# B&R Automation Studio project 8238 (part 31)

### Program Logical/OPCuA_Client/Inwatec (IEC)

#### Variables.var
```iecst
VAR
	i : UINT;
	iw : REFERENCE TO Inwatec_typ;
	iw_d : REFERENCE TO Inwatec_data_typ;
	comm : REFERENCE TO Comm_typ;
	iw_r : REFERENCE TO Inwatec_data_typ;
END_VAR
```

#### Main.st
```iecst
PROGRAM _INIT
//Config and manage inwatec OPCuA communications
Inwatec[1].Config.ServerURL := 'opc.tcp://10.16.118.1:3001';
Inwatec[1].Config.Direction := INWATEC_RELEASE_TO;
Inwatec[1].Config.CommID 		:= 81;

Inwatec[2].Config.ServerURL := 'opc.tcp://10.16.118.1:3002';
Inwatec[2].Config.Direction := INWATEC_RELEASE_TO;
Inwatec[2].Config.CommID 		:= 82;

Inwatec[3].Config.ServerURL := 'opc.tcp://10.16.118.1:3003';
Inwatec[3].Config.Direction := INWATEC_RELEASE_TO;
Inwatec[3].Config.CommID 		:= 83;

Inwatec[4].Config.ServerURL := 'opc.tcp://10.16.118.1:3101';
Inwatec[4].Config.Direction := INWATEC_RECIEVE_FROM;
Inwatec[4].Config.CommID 		:= 84;

Inwatec[5].Config.ServerURL := 'opc.tcp://10.16.118.1:3102';
Inwatec[5].Config.Direction := INWATEC_RECIEVE_FROM;
Inwatec[5].Config.CommID 		:= 85;

Inwatec[6].Config.ServerURL := 'opc.tcp://10.16.118.1:3103';
Inwatec[6].Config.Direction := INWATEC_RECIEVE_FROM;
Inwatec[6].Config.CommID 		:= 86;

Inwatec[7].Config.ServerURL := 'opc.tcp://10.16.118.2:3001';
Inwatec[7].Config.Direction := INWATEC_RELEASE_TO;
Inwatec[7].Config.CommID 		:= 87;

Inwatec[8].Config.ServerURL := 'opc.tcp://10.16.118.2:3002';
Inwatec[8].Config.Direction := INWATEC_RELEASE_TO;
Inwatec[8].Config.CommID 		:= 88;

Inwatec[9].Config.ServerURL := 'opc.tcp://10.16.118.2:3003';
Inwatec[9].Config.Direction := INWATEC_RELEASE_TO;
Inwatec[9].Config.CommID 		:= 89;

Inwatec[10].Config.ServerURL := 'opc.tcp://10.16.118.2:3004';
Inwatec[10].Config.Direction := INWATEC_RELEASE_TO;
Inwatec[10].Config.CommID 		:= 90;

Inwatec[11].Config.ServerURL := 'opc.tcp://10.16.118.2:3101';
Inwatec[11].Config.Direction := INWATEC_RECIEVE_FROM;
Inwatec[11].Config.CommID 		:= 91;

END_PROGRAM

PROGRAM _CYCLIC

FOR i := 1 TO MAX_INWATEC_INTERFACES DO
	iw ACCESS ADR(Inwatec[i]);
	//Range check
	IF (iw.Config.CommID > 0) AND (iw.Config.CommID <= MAX_COMM) THEN
		comm ACCESS ADR(Comm[iw.Config.CommID]);

		CASE iw.Config.Direction OF
			INWATEC_RELEASE_TO:  // We need to set the batch information
				iw_d ACCESS ADR(iw.Outlet);		// Write Vars
				iw_r ACCESS ADR(iw.Inlet);		// Read Vars

				iw_d.batch_id 					:= comm.BatchID;
				iw_d.weight 						:= (UINT_TO_REAL(comm.Weight)/10);
				iw_d.customer_numeric 	:= comm.Customer;
				iw_d.category_numeric		:= comm.Category;
				iw_d.batch_count 				:= comm.Batch_QtyRemaining;

				iw_d.tx_handshake.0 		:= comm.BagReady;				// Bag in position

				// Read Variables
				comm.DropLoad 				:= iw_r.tx_handshake.0;
				comm.Unloading				:= iw_r.tx_handshake.1;
				comm.LoadDropped			:= iw_r.tx_handshake.2;

			INWATEC_RECIEVE_FROM:// We are reading the batch information.
				iw_d ACCESS ADR(iw.Inlet); 		// Write Vars
				iw_r ACCESS ADR(iw.Outlet);		// Read Vars

				iw_d.tx_handshake.0 		:= comm.ReadyToLoad; 	// Bag in position ready for load
				iw_d.tx_handshake.1 		:= comm.Loading;			// Recieving load
				iw_d.tx_handshake.2 		:= comm.LoadRecieved;	// Bag has recieved the load

				// Read Variables
				comm.BatchID 						:= iw_r.batch_id;
				comm.Weight							:= REAL_TO_UINT(iw_r.weight * 10);
				comm.Customer 					:= iw_r.customer_numeric;
				comm.Category						:= iw_r.category_numeric;
				comm.Batch_QtyRemaining	:= iw_r.batch_count;

				comm.ReadyToLoad				:= iw_r.tx_handshake.0;
				comm.Unloading					:= iw_r.tx_handshake.1;
				comm.UnloadFinished			:= iw_r.tx_handshake.2;

			ELSE
				iw_d ACCESS ADR(iw.Inlet);	// Code just ensure we don;t get a pointer error.
				iw_r ACCESS ADR(iw.Outlet);
		END_CASE;

		//Common controls.
		iw_d.system_status.0 := 0;// Is there any alarm on the device;
		iw_d.system_status.1 := 1; // PLC is alive;
		iw_d.system_status.2 := NOT comm.HaltSys; // System is in production (Maybe map Estop zone here)

		iw_d.i_am_alive 			:= Std.Clock1s;

		IF iw_r.i_am_alive THEN
			comm.LiveTime := 500; // 5s ish..
			iw_r.i_am_alive := 0;
		ELSIF (comm.LiveTime > 0) THEN
				comm.LiveTime := (comm.LiveTime - 1);
		END_IF;
		comm.Live := (comm.LiveTime > 0);

	END_IF;
END_FOR;

END_PROGRAM
```

### Program Logical/OPCuA_Client/OPCuAClient (IEC, version 1.00.1)

#### Main.st - Init, cyclic, exit code
```iecst
PROGRAM _INIT

	#if (MAX_OPCuA_CLIENTS < MAX_INWATEC_INTERFACES)
		#error 'Not enough opcua clients for Inwatec'
	#endif

	_inwatec_config;

	////Test connection.
	//OPCuA_Client[3].Config.ServerURL :=	'opc.tcp://10.8.4.20:4840';  // IP Address of interface.
	//
	//OPCuA_Client[3].Config.SessionUser.UserIdentityTokenType := UAUITT_Username;
	//OPCuA_Client[3].Config.SessionUser.TokenParam1 := 'test';  //UserName
	//OPCuA_Client[3].Config.SessionUser.TokenParam2 := 'test';  //Password
	//
	//
	////Set the Vars.
	//OPCuA_Client[3].Config.Data.Read[0].NodeID.Identifier := '::AsGlobalPV:OpcUa.VC[231].Write.Heartbeat';
	//OPCuA_Client[3].Config.Data.Read[0].Variable := 'TestRead[0]';
	//OPCuA_Client[3].Config.Data.Read[1].NodeID.Identifier := '::AsGlobalPV:OpcUa.VC[231].Write.PermissionToMove';
	//OPCuA_Client[3].Config.Data.Read[1].Variable := 'TestRead[1]';
	//OPCuA_Client[3].Config.Data.Read[2].NodeID.Identifier := '::AsGlobalPV:OpcUa.VC[231].Write.ReleaseBag';
	//OPCuA_Client[3].Config.Data.Read[2].Variable := 'TestRead[2]';
	//OPCuA_Client[3].Config.Data.Read[3].NodeID.Identifier := '::AsGlobalPV:OpcUa.VC[231].Write.ReceiveBag';
	//OPCuA_Client[3].Config.Data.Read[3].Variable := 'TestRead[3]';
	//
	//OPCuA_Client[3].Config.Data.Write[0].NodeID.Identifier := '::AsGlobalPV:OpcUa.VC[231].Read.Heartbeat';
	//OPCuA_Client[3].Config.Data.Write[0].Variable := 'TestWrite[0]';
	//OPCuA_Client[3].Config.Data.Write[1].NodeID.Identifier := '::AsGlobalPV:OpcUa.VC[231].Read.Auto';
	//OPCuA_Client[3].Config.Data.Write[1].Variable := 'TestWrite[1]';
	//OPCuA_Client[3].Config.Data.Write[2].NodeID.Identifier := '::AsGlobalPV:OpcUa.VC[231].Read.Manual';
	//OPCuA_Client[3].Config.Data.Write[2].Variable := 'TestWrite[2]';
	//OPCuA_Client[3].Config.Data.Write[3].NodeID.Identifier := '::AsGlobalPV:OpcUa.VC[231].Read.ChuteBlocked';
	//OPCuA_Client[3].Config.Data.Write[3].Variable := 'TestWrite[3]';

	FOR x := 1 TO MAX_OPCuA_CLIENTS DO
		client ACCESS ADR (OPCuA_Client[x]);
		client.Config.SessionInfo.SessionName := 'supertrack';
		client.Config.SessionInfo.ApplicationName := '';
		client.Config.SessionInfo.SecurityMsgMode := UASecurityMsgMode_Sign;//UASecurityMsgMode_BestAvailab;
		client.Config.SessionInfo.SecurityPolicy := UASecurityPolicy_Basic256Sha256;//UASecurityPolicy_BestAvailable;
		client.Config.SessionInfo.CertificateStore := '';
		client.Config.SessionInfo.ClientCertificateName := '';
		client.Config.SessionInfo.ServerUri := '';
		client.Config.SessionInfo.CheckServerCertificate := 0;
		client.Config.SessionInfo.TransportProfile := UATP_UATcp;
		client.Config.SessionInfo.UserIdentityToken := client.Config.SessionUser;
		client.Config.SessionInfo.VendorSpecificParameter := '';
		client.Config.SessionInfo.SessionTimeout := T#5s;
		client.Config.SessionInfo.MonitorConnection := T#500ms;
		//client.Config.SessionInfo.LocaleIDs

		client.Config.Data.ReadCount := MAX_READ_NODES;
		FOR i := 0 TO MAX_READ_NODES DO
			client.Config.Data.Read[i].NodeID.IdentifierType := UAIdentifierType_String;
			client.Config.Data.Read[i].NodeInfo.AttributeId := UAAI_Value;
			IF (client.Config.Data.Read[i].NodeID.Identifier = '') THEN
				client.Config.Data.ReadCount := i;
				EXIT;
			END_IF;
		END_FOR;

		client.Config.Data.WriteCount := MAX_WRITE_NODES;
		FOR i := 0 TO MAX_WRITE_NODES DO
			client.Config.Data.Write[i].NodeID.IdentifierType := UAIdentifierType_String;
			client.Config.Data.Write[i].NodeInfo.AttributeId := UAAI_Value;
			IF (client.Config.Data.Write[i].NodeID.Identifier = '') THEN
				client.Config.Data.WriteCount := i;
				EXIT;
			END_IF;
		END_FOR;

		client.Functions.RetryTimer.PT := T#5s; // Time to try to reconnect if the server isn;t available.
	END_FOR;

END_PROGRAM

PROGRAM _CYCLIC
//MAX of 40 Connections.

	FOR x := 1 TO MAX_OPCuA_CLIENTS DO
		client ACCESS ADR (OPCuA_Client[x]);
		f ACCESS ADR(client.Functions);
		IF client.Config.ServerURL <> '' THEN

			f.Connect.Execute 			:= (client.State = OPCuA_CLIENT_STATE_CONNECT);
			f.GetNameSpace.Execute	:= (client.State = OPCuA_CLIENT_STATE_GET_NAMESPACE);
			f.ReadBulk.Execute := f.WriteBulk.Execute	:= (client.State = OPCuA_CLIENT_STATE_READ_WRITE);
			f.Disconnect.Execute 		:= (client.State = OPCuA_CLIENT_STATE_DISCONNECT);

			CASE client.State OF

				OPCuA_CLIENT_STATE_CONNECT:
					f.Connect.ServerEndpointUrl := client.Config.ServerURL;
					f.Connect.SessionConnectInfo := client.Config.SessionInfo;
					f.Connect.Timeout := T#1s;
					IF f.Connect.Done THEN
						client.State := OPCuA_CLIENT_STATE_GET_NAMESPACE;
					ELSIF f.Connect.Error THEN
						client.Error.ErrorState := client.State;
						client.State := OPCuA_CLIENT_STATE_ERROR;
						client.Error.ErrorID :=  f.Connect.ErrorID;
					END_IF;

				OPCuA_CLIENT_STATE_GET_NAMESPACE:
					f.GetNameSpace.ConnectionHdl  := f.Connect.ConnectionHdl;
					f.GetNameSpace.NamespaceUri		:= 'urn:B&R/pv/';
					f.GetNameSpace.Timeout 				:= T#1s;

					IF f.GetNameSpace.Done THEN
						client.State := OPCuA_CLIENT_STATE_BUILD_DATA;
					ELSIF f.GetNameSpace.Error THEN
						client.Error.ErrorState := client.State;
						client.State := OPCuA_CLIENT_STATE_ERROR;
						client.Error.ErrorID :=  f.GetNameSpace.ErrorID;
					END_IF;

				OPCuA_CLIENT_STATE_BUILD_DATA:

					FOR i := 0 TO client.Config.Data.ReadCount DO
						client.ReadData.NodeID[i].NamespaceIndex 	:= f.GetNameSpace.NamespaceIndex;
						client.ReadData.NodeID[i].IdentifierType 	:= client.Config.Data.Read[i].NodeID.IdentifierType;
						client.ReadData.NodeID[i].Identifier 			:= client.Config.Data.Read[i].NodeID.Identifier;
						client.ReadData.NodeInfo[i].AttributeId 	:= client.Config.Data.Read[i].NodeInfo.AttributeId;
						client.ReadData.Variable[i]								:= client.Config.Data.Read[i].Variable;
					END_FOR;

					FOR i := 0 TO client.Config.Data.WriteCount DO
						client.WriteData.NodeID[i].NamespaceIndex 	:= f.GetNameSpace.NamespaceIndex;
						client.WriteData.NodeID[i].IdentifierType 	:= client.Config.Data.Write[i].NodeID.IdentifierType;
						client.WriteData.NodeID[i].Identifier 			:= client.Config.Data.Write[i].NodeID.Identifier;
						client.WriteData.NodeInfo[i].AttributeId 		:= client.Config.Data.Write[i].NodeInfo.AttributeId;
						client.WriteData.Variable[i]								:= client.Config.Data.Write[i].Variable;

					END_FOR;

					client.State := OPCuA_CLIENT_STATE_READ_WRITE;

				OPCuA_CLIENT_STATE_READ_WRITE:
					f.ReadBulk.ConnectionHdl 	:= f.Connect.ConnectionHdl;
					f.ReadBulk.NodeIDCount 		:= client.Config.Data.ReadCount;
					f.ReadBulk.NodeAddInfo 		:= ADR(client.ReadData.NodeInfo);
					f.ReadBulk.NodeErrorIDs 	:= ADR(client.ReadData.ErrorID);
					f.ReadBulk.NodeIDs 				:= ADR(client.ReadData.NodeID);
					f.ReadBulk.TimeStamps 		:= ADR(client.ReadData.TimeStamps);
					f.ReadBulk.Variables 			:= ADR(client.ReadData.Variable);
					f.ReadBulk.Timeout 				:= T#1500ms;
					IF f.ReadBulk.Done THEN
						f.ReadBulk.Execute := 0; // Read Cyclica
						f.ReadBulk;
					ELSIF f.ReadBulk.Error THEN
						IF 	f.ReadBulk.ErrorID = OPCuA_ERR_OUT_OF_SERVICE THEN
							client.State := OPCuA_CLIENT_STATE_DISCONNECT;
						ELSE
							client.Error.ErrorState := client.State;
							client.State := OPCuA_CLIENT_STATE_ERROR;
							IF (f.ReadBulk.ErrorID > 0) THEN
								client.Error.ErrorID := f.ReadBulk.ErrorID;
							ELSE
								//Look for the bad node..
								FOR i := 0 TO client.Config.Data.ReadCount DO
									IF (client.ReadData.ErrorID[i] > 0) THEN
										client.Error.ErrorID := client.ReadData.ErrorID[i];
										client.Error.ErrorNode := i;
										EXIT;
									END_IF;
								END_FOR;
							END_IF;
						END_IF;

					END_IF

					//Disadvantage of writing like this, is we are always pushing just like tradional TCP.
					f.WriteBulk.ConnectionHdl := f.Connect.ConnectionHdl;
					f.WriteBulk.NodeIDCount		:= client.Config.Data.WriteCount;
					f.WriteBulk.NodeAddInfo		:= ADR(client.WriteData.NodeInfo);
					f.WriteBulk.NodeErrorIDs	:= ADR(client.WriteData.ErrorID);
					f.WriteBulk.NodeIDs				:= ADR(client.WriteData.NodeID);
					f.WriteBulk.Variables			:= ADR(client.WriteData.Variable);
					f.WriteBulk.Timeout				:= T#1500ms;

					IF f.WriteBulk.Done THEN
						f.WriteBulk.Execute := 0; // Read Cyclica
						f.WriteBulk();
					ELSIF f.WriteBulk.Error THEN
						IF 	f.WriteBulk.ErrorID = OPCuA_ERR_OUT_OF_SERVICE THEN
							client.State := OPCuA_CLIENT_STATE_DISCONNECT;
						ELSE
							client.Error.ErrorState := OPCuA_CLIENT_STATE_READ_WRITE + 1000;// Add 1000 to show its a write failure.
							client.State := OPCuA_CLIENT_STATE_ERROR;
							IF (f.WriteBulk.ErrorID > 0) THEN
								client.Error.ErrorID := f.WriteBulk.ErrorID;
							ELSE
								//Look for the bad node..
								FOR i := 0 TO client.Config.Data.WriteCount DO
									IF (client.WriteData.ErrorID[i] > 0) THEN
										client.Error.ErrorID := client.WriteData.ErrorID[i];
										client.Error.ErrorNode := i;
										EXIT;
									END_IF;
								END_FOR;
							END_IF;
						END_IF;

					END_IF;

				OPCuA_CLIENT_STATE_DISCONNECT:
					f.Disconnect.ConnectionHdl := f.Connect.ConnectionHdl;
					f.Disconnect.Timeout := T#2s;
					IF f.Disconnect.Done THEN
						client.State := OPCuA_CLIENT_STATE_CONNECT;
					ELSIF f.Disconnect.Error THEN
						IF (f.Connect.ConnectionHdl = 0) OR (f.Disconnect.ErrorID = 16#A0080000) OR (f.Disconnect.ErrorID = 16#80AD0000)  THEN
							client.State := OPCuA_CLIENT_STATE_CONNECT;
						ELSE
							//client.State := OPCuA_CLIENT_STATE_ERROR;
							//client.Error.ErrorID := f.Disconnect.ErrorID;
						END_IF;
					END_IF;

				OPCuA_CLIENT_STATE_ERROR:
					//Maybe should just write to a logger then restart!
					IF client.Functions.RetryTimer.Q THEN
						IF (f.Connect.ConnectionHdl > 0) THEN
							client.State := OPCuA_CLIENT_STATE_DISCONNECT; // Always try to disconnect any open connections before reconnecting.
						ELSE
							client.State := OPCuA_CLIENT_STATE_CONNECT;
						END_IF;
					ELSIF (client.Error.ErrorID = OPCuA_ERR_TIMEOUT) THEN
						//				client.Functions.RetryTimer.IN := 1;
						//			ELSE
						//				client.State := OPCuA_CLIENT_STATE_DISCONNECT;
					END_IF;

			END_CASE;
			client.Functions.ErrorStatePLS.CLK := (client.State = OPCuA_CLIENT_STATE_ERROR);
			client.Functions.ErrorStatePLS();

			IF client.Functions.ErrorStatePLS.Q THEN
				brsmemcpy(ADR(client.Error.ErrorCode),ADR(client.Error.ErrorID) + 2,2);
				getErrorText.ErrorID := client.Error.ErrorCode;
				getErrorText();
				client.Error.Message := 	getErrorText.ErrorMessage;
			END_IF;

			f.Connect();
			f.GetNameSpace();
			f.ReadBulk();
			f.WriteBulk();
			f.Disconnect();
			client.Functions.RetryTimer.IN := (client.State = OPCuA_CLIENT_STATE_ERROR);
			client.Functions.RetryTimer();
		//client.Functions.RetryTimer.IN := 0;
		END_IF;
	END_FOR;
	//TestRead;//
	//TestWrite;
	//	TestReadx;//
	//	TestWritex;

END_PROGRAM

PROGRAM _EXIT
(* Insert code here *)

END_PROGRAM
```

#### inwatec.st - *Special config for building inwatec interfaces
```iecst
ACTION _inwatec_config:

FOR i := 1 TO MAX_INWATEC_INTERFACES DO
	//Always match the inwatec array to the opcua array
	iw ACCESS ADR(Inwatec[i]);
	client ACCESS ADR(OPCuA_Client[i]);

	client.Config.ServerURL :=	iw.Config.ServerURL;
	client.Config.SessionUser := iw.Config.Authenication;

	CASE iw.Config.Direction OF
		0: //Dropping onto Inwatec
			//Write to Outlet, Read from Inlet

			client.Config.Data.Read[0].NodeID.Identifier := '::BatchIn:batch_to_inwatec[0].inlet.batch_count';
			client.Config.Data.Read[1].NodeID.Identifier := '::BatchIn:batch_to_inwatec[0].inlet.batch_id';
			client.Config.Data.Read[2].NodeID.Identifier := '::BatchIn:batch_to_inwatec[0].inlet.category';
			client.Config.Data.Read[3].NodeID.Identifier := '::BatchIn:batch_to_inwatec[0].inlet.category_name';
			client.Config.Data.Read[4].NodeID.Identifier := '::BatchIn:batch_to_inwatec[0].inlet.category_numeric';
			client.Config.Data.Read[5].NodeID.Identifier := '::BatchIn:batch_to_inwatec[0].inlet.customer';
			client.Config.Data.Read[6].NodeID.Identifier := '::BatchIn:batch_to_inwatec[0].inlet.customer_name';
			client.Config.Data.Read[7].NodeID.Identifier := '::BatchIn:batch_to_inwatec[0].inlet.customer_numeric';
			client.Config.Data.Read[8].NodeID.Identifier := '::BatchIn:batch_to_inwatec[0].inlet.i_am_alive';
			client.Config.Data.Read[9].NodeID.Identifier := '::BatchIn:batch_to_inwatec[0].inlet.lot';
			client.Config.Data.Read[10].NodeID.Identifier := '::BatchIn:batch_to_inwatec[0].inlet.lot_numeric';
			client.Config.Data.Read[11].NodeID.Identifier := '::BatchIn:batch_to_inwatec[0].inlet.option_1';
			client.Config.Data.Read[12].NodeID.Identifier := '::BatchIn:batch_to_inwatec[0].inlet.option_2';
			client.Config.Data.Read[13].NodeID.Identifier := '::BatchIn:batch_to_inwatec[0].inlet.source_id';
			client.Config.Data.Read[14].NodeID.Identifier := '::BatchIn:batch_to_inwatec[0].inlet.sublot';
			client.Config.Data.Read[15].NodeID.Identifier := '::BatchIn:batch_to_inwatec[0].inlet.sublot_numeric';
			client.Config.Data.Read[16].NodeID.Identifier := '::BatchIn:batch_to_inwatec[0].inlet.system_status';
			client.Config.Data.Read[17].NodeID.Identifier := '::BatchIn:batch_to_inwatec[0].inlet.tx_handshake';
			client.Config.Data.Read[18].NodeID.Identifier := '::BatchIn:batch_to_inwatec[0].inlet.weight';
			client.Config.Data.Read[19].NodeID.Identifier := '::BatchIn:batch_to_inwatec[0].inlet.option_flag_1';
			client.Config.Data.Read[20].NodeID.Identifier := '::BatchIn:batch_to_inwatec[0].inlet.option_flag_2';

			client.Config.Data.Write[0].NodeID.Identifier := '::BatchIn:batch_to_inwatec[0].outlet.batch_count';
			client.Config.Data.Write[1].NodeID.Identifier := '::BatchIn:batch_to_inwatec[0].outlet.batch_id';
			client.Config.Data.Write[2].NodeID.Identifier := '::BatchIn:batch_to_inwatec[0].outlet.category';
			client.Config.Data.Write[3].NodeID.Identifier := '::BatchIn:batch_to_inwatec[0].outlet.category_name';
			client.Config.Data.Write[4].NodeID.Identifier := '::BatchIn:batch_to_inwatec[0].outlet.category_numeric';
			client.Config.Data.Write[5].NodeID.Identifier := '::BatchIn:batch_to_inwatec[0].outlet.customer';
			client.Config.Data.Write[6].NodeID.Identifier := '::BatchIn:batch_to_inwatec[0].outlet.customer_name';
			client.Config.Data.Write[7].NodeID.Identifier := '::BatchIn:batch_to_inwatec[0].outlet.customer_numeric';
			client.Config.Data.Write[8].NodeID.Identifier := '::BatchIn:batch_to_inwatec[0].outlet.i_am_alive';
			client.Config.Data.Write[9].NodeID.Identifier := '::BatchIn:batch_to_inwatec[0].outlet.lot';
			client.Config.Data.Write[10].NodeID.Identifier := '::BatchIn:batch_to_inwatec[0].outlet.lot_numeric';
			client.Config.Data.Write[11].NodeID.Identifier := '::BatchIn:batch_to_inwatec[0].outlet.option_1';
			client.Config.Data.Write[12].NodeID.Identifier := '::BatchIn:batch_to_inwatec[0].outlet.option_2';
			client.Config.Data.Write[13].NodeID.Identifier := '::BatchIn:batch_to_inwatec[0].outlet.source_id';
			client.Config.Data.Write[14].NodeID.Identifier := '::BatchIn:batch_to_inwatec[0].outlet.sublot';
			client.Config.Data.Write[15].NodeID.Identifier := '::BatchIn:batch_to_inwatec[0].outlet.sublot_numeric';
			client.Config.Data.Write[16].NodeID.Identifier := '::BatchIn:batch_to_inwatec[0].outlet.system_status';
			client.Config.Data.Write[17].NodeID.Identifier := '::BatchIn:batch_to_inwatec[0].outlet.tx_handshake';
			client.Config.Data.Write[18].NodeID.Identifier := '::BatchIn:batch_to_inwatec[0].outlet.weight';
			client.Config.Data.Write[19].NodeID.Identifier := '::BatchIn:batch_to_inwatec[0].outlet.option_flag_1';
			client.Config.Data.Write[20].NodeID.Identifier := '::BatchIn:batch_to_inwatec[0].outlet.option_flag_2';

			brsitoa(i,ADR(str_index));
			FOR x := 0 TO MAX_READ_NODES DO
				client.Config.Data.Read[x].Variable := 'Inwatec[';
				brsstrcat(ADR(client.Config.Data.Read[x].Variable),ADR(str_index));
			END_FOR;
			brsstrcat(ADR(client.Config.Data.Read[0].Variable),ADR('].Inlet.batch_count'));
			brsstrcat(ADR(client.Config.Data.Read[1].Variable),ADR('].Inlet.batch_id'));
			brsstrcat(ADR(client.Config.Data.Read[2].Variable),ADR('].Inlet.category'));
			brsstrcat(ADR(client.Config.Data.Read[3].Variable),ADR('].Inlet.category_name'));
			brsstrcat(ADR(client.Config.Data.Read[4].Variable),ADR('].Inlet.category_numeric'));
			brsstrcat(ADR(client.Config.Data.Read[5].Variable),ADR('].Inlet.customer'));
			brsstrcat(ADR(client.Config.Data.Read[6].Variable),ADR('].Inlet.customer_name'));
			brsstrcat(ADR(client.Config.Data.Read[7].Variable),ADR('].Inlet.customer_numeric'));
			brsstrcat(ADR(client.Config.Data.Read[8].Variable),ADR('].Inlet.i_am_alive'));
			brsstrcat(ADR(client.Config.Data.Read[9].Variable),ADR('].Inlet.lot'));
			brsstrcat(ADR(client.Config.Data.Read[10].Variable),ADR('].Inlet.lot_numeric'));
			brsstrcat(ADR(client.Config.Data.Read[11].Variable),ADR('].Inlet.option_1'));
			brsstrcat(ADR(client.Config.Data.Read[12].Variable),ADR('].Inlet.option_2'));
			brsstrcat(ADR(client.Config.Data.Read[13].Variable),ADR('].Inlet.source_id'));
			brsstrcat(ADR(client.Config.Data.Read[14].Variable),ADR('].Inlet.sublot'));
			brsstrcat(ADR(client.Config.Data.Read[15].Variable),ADR('].Inlet.sublot_numeric'));
			brsstrcat(ADR(client.Config.Data.Read[16].Variable),ADR('].Inlet.system_status'));
			brsstrcat(ADR(client.Config.Data.Read[17].Variable),ADR('].Inlet.tx_handshake'));
			brsstrcat(ADR(client.Config.Data.Read[18].Variable),ADR('].Inlet.weight'));
			brsstrcat(ADR(client.Config.Data.Read[19].Variable),ADR('].Inlet.option_flag_1'));
			brsstrcat(ADR(client.Config.Data.Read[20].Variable),ADR('].Inlet.option_flag_2'));

			brsitoa(i,ADR(str_index));
			FOR x := 0 TO MAX_WRITE_NODES DO
				client.Config.Data.Read[x].Variable := 'Inwatec[';
				brsstrcat(ADR(client.Config.Data.Read[x].Variable),ADR(str_index));
			END_FOR;
			brsstrcat(ADR(client.Config.Data.Write[0].Variable),ADR('].Outlet.batch_count'));
			brsstrcat(ADR(client.Config.Data.Write[1].Variable),ADR('].Outlet.batch_id'));
			brsstrcat(ADR(client.Config.Data.Write[2].Variable),ADR('].Outlet.category'));
			brsstrcat(ADR(client.Config.Data.Write[3].Variable),ADR('].Outlet.category_name'));
			brsstrcat(ADR(client.Config.Data.Write[4].Variable),ADR('].Outlet.category_numeric'));
			brsstrcat(ADR(client.Config.Data.Write[5].Variable),ADR('].Outlet.customer'));
			brsstrcat(ADR(client.Config.Data.Write[6].Variable),ADR('].Outlet.customer_name'));
			brsstrcat(ADR(client.Config.Data.Write[7].Variable),ADR('].Outlet.customer_numeric'));
			brsstrcat(ADR(client.Config.Data.Write[8].Variable),ADR('].Outlet.i_am_alive'));
			brsstrcat(ADR(client.Config.Data.Write[9].Variable),ADR('].Outlet.lot'));
			brsstrcat(ADR(client.Config.Data.Write[10].Variable),ADR('].Outlet.lot_numeric'));
			brsstrcat(ADR(client.Config.Data.Write[11].Variable),ADR('].Outlet.option_1'));
			brsstrcat(ADR(client.Config.Data.Write[12].Variable),ADR('].Outlet.option_2'));
			brsstrcat(ADR(client.Config.Data.Write[13].Variable),ADR('].Outlet.source_id'));
			brsstrcat(ADR(client.Config.Data.Write[14].Variable),ADR('].Outlet.sublot'));
			brsstrcat(ADR(client.Config.Data.Write[15].Variable),ADR('].Outlet.sublot_numeric'));
			brsstrcat(ADR(client.Config.Data.Write[16].Variable),ADR('].Outlet.system_status'));
			brsstrcat(ADR(client.Config.Data.Write[17].Variable),ADR('].Outlet.tx_handshake'));
			brsstrcat(ADR(client.Config.Data.Write[18].Variable),ADR('].Outlet.weight'));
			brsstrcat(ADR(client.Config.Data.Write[19].Variable),ADR('].Outlet.option_flag_1'));
			brsstrcat(ADR(client.Config.Data.Write[20].Variable),ADR('].Outlet.option_flag_2'));

		1: //Recieving from Inwatec
				//Write to Inlet, Read from Outlet
				client.Config.Data.Read[0].NodeID.Identifier := '::BatchOut:batch_from_inwatec[0].outlet.batch_count';
				client.Config.Data.Read[1].NodeID.Identifier := '::BatchOut:batch_from_inwatec[0].outlet.batch_id';
				client.Config.Data.Read[2].NodeID.Identifier := '::BatchOut:batch_from_inwatec[0].outlet.category';
				client.Config.Data.Read[3].NodeID.Identifier := '::BatchOut:batch_from_inwatec[0].outlet.category_name';
				client.Config.Data.Read[4].NodeID.Identifier := '::BatchOut:batch_from_inwatec[0].outlet.category_numeric';
				client.Config.Data.Read[5].NodeID.Identifier := '::BatchOut:batch_from_inwatec[0].outlet.customer';
				client.Config.Data.Read[6].NodeID.Identifier := '::BatchOut:batch_from_inwatec[0].outlet.customer_name';
				client.Config.Data.Read[7].NodeID.Identifier := '::BatchOut:batch_from_inwatec[0].outlet.customer_numeric';
				client.Config.Data.Read[8].NodeID.Identifier := '::BatchOut:batch_from_inwatec[0].outlet.i_am_alive';
				client.Config.Data.Read[9].NodeID.Identifier := '::BatchOut:batch_from_inwatec[0].outlet.lot';
				client.Config.Data.Read[10].NodeID.Identifier := '::BatchOut:batch_from_inwatec[0].outlet.lot_numeric';
				client.Config.Data.Read[11].NodeID.Identifier := '::BatchOut:batch_from_inwatec[0].outlet.option_1';
				client.Config.Data.Read[12].NodeID.Identifier := '::BatchOut:batch_from_inwatec[0].outlet.option_2';
				client.Config.Data.Read[13].NodeID.Identifier := '::BatchOut:batch_from_inwatec[0].outlet.source_id';
				client.Config.Data.Read[14].NodeID.Identifier := '::BatchOut:batch_from_inwatec[0].outlet.sublot';
				client.Config.Data.Read[15].NodeID.Identifier := '::BatchOut:batch_from_inwatec[0].outlet.sublot_numeric';
				client.Config.Data.Read[16].NodeID.Identifier := '::BatchOut:batch_from_inwatec[0].outlet.system_status';
				client.Config.Data.Read[17].NodeID.Identifier := '::BatchOut:batch_from_inwatec[0].outlet.tx_handshake';
				client.Config.Data.Read[18].NodeID.Identifier := '::BatchOut:batch_from_inwatec[0].outlet.weight';
				client.Config.Data.Read[19].NodeID.Identifier := '::BatchOut:batch_from_inwatec[0].outlet.option_flag_1';
				client.Config.Data.Read[20].NodeID.Identifier := '::BatchOut:batch_from_inwatec[0].outlet.option_flag_2';

				client.Config.Data.Write[0].NodeID.Identifier := '::BatchOut:batch_from_inwatec[0].inlet.batch_count';
				client.Config.Data.Write[1].NodeID.Identifier := '::BatchOut:batch_from_inwatec[0].inlet.batch_id';
				client.Config.Data.Write[2].NodeID.Identifier := '::BatchOut:batch_from_inwatec[0].inlet.category';
				client.Config.Data.Write[3].NodeID.Identifier := '::BatchOut:batch_from_inwatec[0].inlet.category_name';
				client.Config.Data.Write[4].NodeID.Identifier := '::BatchOut:batch_from_inwatec[0].inlet.category_numeric';
				client.Config.Data.Write[5].NodeID.Identifier := '::BatchOut:batch_from_inwatec[0].inlet.customer';
				client.Config.Data.Write[6].NodeID.Identifier := '::BatchOut:batch_from_inwatec[0].inlet.customer_name';
				client.Config.Data.Write[7].NodeID.Identifier := '::BatchOut:batch_from_inwatec[0].inlet.customer_numeric';
				client.Config.Data.Write[8].NodeID.Identifier := '::BatchOut:batch_from_inwatec[0].inlet.i_am_alive';
				client.Config.Data.Write[9].NodeID.Identifier := '::BatchOut:batch_from_inwatec[0].inlet.lot';
				client.Config.Data.Write[10].NodeID.Identifier := '::BatchOut:batch_from_inwatec[0].inlet.lot_numeric';
				client.Config.Data.Write[11].NodeID.Identifier := '::BatchOut:batch_from_inwatec[0].inlet.option_1';
				client.Config.Data.Write[12].NodeID.Identifier := '::BatchOut:batch_from_inwatec[0].inlet.option_2';
				client.Config.Data.Write[13].NodeID.Identifier := '::BatchOut:batch_from_inwatec[0].inlet.source_id';
				client.Config.Data.Write[14].NodeID.Identifier := '::BatchOut:batch_from_inwatec[0].inlet.sublot';
				client.Config.Data.Write[15].NodeID.Identifier := '::BatchOut:batch_from_inwatec[0].inlet.sublot_numeric';
				client.Config.Data.Write[16].NodeID.Identifier := '::BatchOut:batch_from_inwatec[0].inlet.system_status';
				client.Config.Data.Write[17].NodeID.Identifier := '::BatchOut:batch_from_inwatec[0].inlet.tx_handshake';
				client.Config.Data.Write[18].NodeID.Identifier := '::BatchOut:batch_from_inwatec[0].inlet.weight';
				client.Config.Data.Write[19].NodeID.Identifier := '::BatchOut:batch_from_inwatec[0].inlet.option_flag_1';
				client.Config.Data.Write[20].NodeID.Identifier := '::BatchOut:batch_from_inwatec[0].inlet.option_flag_2';

				brsitoa(i,ADR(str_index));
				FOR x := 0 TO MAX_READ_NODES DO
					client.Config.Data.Read[x].Variable := 'Inwatec[';
					brsstrcat(ADR(client.Config.Data.Read[x].Variable),ADR(str_index));
				END_FOR;
				brsstrcat(ADR(client.Config.Data.Read[0].Variable),ADR('].Outlet.batch_count'));
				brsstrcat(ADR(client.Config.Data.Read[1].Variable),ADR('].Outlet.batch_id'));
				brsstrcat(ADR(client.Config.Data.Read[2].Variable),ADR('].Outlet.category'));
				brsstrcat(ADR(client.Config.Data.Read[3].Variable),ADR('].Outlet.category_name'));
				brsstrcat(ADR(client.Config.Data.Read[4].Variable),ADR('].Outlet.category_numeric'));
				brsstrcat(ADR(client.Config.Data.Read[5].Variable),ADR('].Outlet.customer'));
				brsstrcat(ADR(client.Config.Data.Read[6].Variable),ADR('].Outlet.customer_name'));
				brsstrcat(ADR(client.Config.Data.Read[7].Variable),ADR('].Outlet.customer_numeric'));
				brsstrcat(ADR(client.Config.Data.Read[8].Variable),ADR('].Outlet.i_am_alive'));
				brsstrcat(ADR(client.Config.Data.Read[9].Variable),ADR('].Outlet.lot'));
				brsstrcat(ADR(client.Config.Data.Read[10].Variable),ADR('].Outlet.lot_numeric'));
				brsstrcat(ADR(client.Config.Data.Read[11].Variable),ADR('].Outlet.option_1'));
				brsstrcat(ADR(client.Config.Data.Read[12].Variable),ADR('].Outlet.option_2'));
				brsstrcat(ADR(client.Config.Data.Read[13].Variable),ADR('].Outlet.source_id'));
				brsstrcat(ADR(client.Config.Data.Read[14].Variable),ADR('].Outlet.sublot'));
				brsstrcat(ADR(client.Config.Data.Read[15].Variable),ADR('].Outlet.sublot_numeric'));
				brsstrcat(ADR(client.Config.Data.Read[16].Variable),ADR('].Outlet.system_status'));
				brsstrcat(ADR(client.Config.Data.Read[17].Variable),ADR('].Outlet.tx_handshake'));
				brsstrcat(ADR(client.Config.Data.Read[18].Variable),ADR('].Outlet.weight'));
				brsstrcat(ADR(client.Config.Data.Read[19].Variable),ADR('].Outlet.option_flag_1'));
				brsstrcat(ADR(client.Config.Data.Read[20].Variable),ADR('].Outlet.option_flag_2'));

				brsitoa(i,ADR(str_index));
				FOR x := 0 TO MAX_WRITE_NODES DO
					client.Config.Data.Read[x].Variable := 'Inwatec[';
					brsstrcat(ADR(client.Config.Data.Read[x].Variable),ADR(str_index));
				END_FOR;
				brsstrcat(ADR(client.Config.Data.Write[0].Variable),ADR('].Inlet.batch_count'));
				brsstrcat(ADR(client.Config.Data.Write[1].Variable),ADR('].Inlet.batch_id'));
				brsstrcat(ADR(client.Config.Data.Write[2].Variable),ADR('].Inlet.category'));
				brsstrcat(ADR(client.Config.Data.Write[3].Variable),ADR('].Inlet.category_name'));
				brsstrcat(ADR(client.Config.Data.Write[4].Variable),ADR('].Inlet.category_numeric'));
				brsstrcat(ADR(client.Config.Data.Write[5].Variable),ADR('].Inlet.customer'));
				brsstrcat(ADR(client.Config.Data.Write[6].Variable),ADR('].Inlet.customer_name'));
				brsstrcat(ADR(client.Config.Data.Write[7].Variable),ADR('].Inlet.customer_numeric'));
				brsstrcat(ADR(client.Config.Data.Write[8].Variable),ADR('].Inlet.i_am_alive'));
				brsstrcat(ADR(client.Config.Data.Write[9].Variable),ADR('].Inlet.lot'));
				brsstrcat(ADR(client.Config.Data.Write[10].Variable),ADR('].Inlet.lot_numeric'));
				brsstrcat(ADR(client.Config.Data.Write[11].Variable),ADR('].Inlet.option_1'));
				brsstrcat(ADR(client.Config.Data.Write[12].Variable),ADR('].Inlet.option_2'));
				brsstrcat(ADR(client.Config.Data.Write[13].Variable),ADR('].Inlet.source_id'));
				brsstrcat(ADR(client.Config.Data.Write[14].Variable),ADR('].Inlet.sublot'));
				brsstrcat(ADR(client.Config.Data.Write[15].Variable),ADR('].Inlet.sublot_numeric'));
				brsstrcat(ADR(client.Config.Data.Write[16].Variable),ADR('].Inlet.system_status'));
				brsstrcat(ADR(client.Config.Data.Write[17].Variable),ADR('].Inlet.tx_handshake'));
				brsstrcat(ADR(client.Config.Data.Write[18].Variable),ADR('].Inlet.weight'));
				brsstrcat(ADR(client.Config.Data.Write[19].Variable),ADR('].Inlet.option_flag_1'));
				brsstrcat(ADR(client.Config.Data.Write[20].Variable),ADR('].Inlet.option_flag_2'));

		END_CASE;

END_FOR;

END_ACTION
```

#### Variables.var - Local variables
```iecst
VAR
	f : REFERENCE TO OPCuaClient_Functions_typ;
	client : REFERENCE TO OPCuaClient_typ;
	i : UINT;
	getErrorText : OPCuaGetErrorMessage;
	x : UINT;
	iw : REFERENCE TO Inwatec_typ;
	str_index : STRING[5];
END_VAR
```

### Library Logical/OPCuA_Client/OPCuAClnt (IEC)
Depends on: AsOpcUac

#### OPCuAClnt.fun - Exported functions and function blocks
```iecst
{REDUND_OK} FUNCTION_BLOCK OPCuaGetErrorMessage (*Returns Text for OPCuA Error ID*) (*$GROUP=User,$CAT=User,$GROUPICON=User.png,$CATICON=User.png*)
	VAR_INPUT
		ErrorID : UDINT;
	END_VAR
	VAR_OUTPUT
		ErrorMessage : STRING[254];
	END_VAR
END_FUNCTION_BLOCK
```

#### GetErrorMessage.st
```iecst
(* Returns Text for OPCuA Error ID *)
FUNCTION_BLOCK OPCuaGetErrorMessage

	CASE ErrorID OF

		16#8000:
			ErrorMessage := 'Unspecified error';
		16#8001:
			ErrorMessage := 'An unexpected error occurred ';
		16#8002:
			ErrorMessage := 'An internal error occurred as a result of a programming or configuration errors.';
		16#8003:
			ErrorMessage := 'Not enough memory to complete the operation.';
		16#8004:
			ErrorMessage := 'An operating system resource is not available';
		16#8005:
			ErrorMessage := 'A low level communication error occurred.';
		16#8006:
			ErrorMessage := 'Encoding halted because of invalid data in the objects being serialized.';
		16#8007:
			ErrorMessage := 'Decoding halted because of invalid data in the stream.';
		16#8008:
			ErrorMessage := 'The message encoding/decoding limits have been exceeded.';
		16#8009:
			ErrorMessage := 'An unrecognized response was received from the server.';
		16#800A:
			ErrorMessage := 'The operation timed out.';
		16#800B:
			ErrorMessage := 'The server does not support the requested service.';
		16#800C:
			ErrorMessage := 'The operation was canceled because the application is shutting down.';
		16#800D:
			ErrorMessage := 'The operation could not complete because the client is not connected to the server.';
		16#800E:
			ErrorMessage := 'The server has stopped and cannot process any requests.';
		16#800F:
			ErrorMessage := 'There was nothing to do because the client passed a list of operations with no elements';

		16#8010:
			ErrorMessage := 'The request could not be processed because it specified too many operations.';
		16#8011:
			ErrorMessage := 'The extension object cannot be (de)serialized because the data type ID is not recognized.';
		16#8012:
			ErrorMessage := 'The certificate provided as a parameter is not valid.';
		16#8013:
			ErrorMessage := 'An error occurred while verifying security.';
		16#8014:
			ErrorMessage := 'The certificate has expired or is not yet valid.';
		16#8015:
			ErrorMessage := 'An issuer certificate has expired or is not yet valid.';
		16#8016:
			ErrorMessage := 'The hostname used to connect to a Server does not match a hostname in the certificate.';
		16#8017:
			ErrorMessage := 'The URI specified in the application description does not match the URI in the certificate.';
		16#8018:
			ErrorMessage := 'The certificate cannot be used for the requested operation.';
		16#8019:
			ErrorMessage := 'The issuer certificate may not be used for the requested operation';
		16#801A:
			ErrorMessage := 'The certificate is not trusted.';
		16#801B:
			ErrorMessage := 'It was not possible to determine if the certificate has been revoked.';
		16#801C:
			ErrorMessage := 'It was not possible to determine if the issuer certificate has been revoked.';
		16#801D:
			ErrorMessage := 'The certificate has been revoked.';
		16#801E:
			ErrorMessage := 'The issuer certificate has been revoked.';
		16#801F:
			ErrorMessage := 'User does not have permission to perform the requested operation';

		16#8020:
			ErrorMessage := 'The user identity token is not valid.';
		16#8021:
			ErrorMessage := 'The user identity token is valid but the server has rejected it.';
		16#8022:
			ErrorMessage := 'The specified secure channel is no longer valid.';
		16#8023:
			ErrorMessage := 'The timestamp is outside the range permitted by the server.';
		16#8024:
			ErrorMessage := ' The nonce does not appear to be a random value or it is not the correct length. ';
		16#8025:
			ErrorMessage := 'The session ID is not valid.';
		16#8026:
			ErrorMessage := 'The session was closed by the client.';
		16#8027:
			ErrorMessage := ' The session cannot be used because ActivateSession has not been called.';
		16#8028:
			ErrorMessage := 'The subscription ID is not valid';
//		16#8029:
//		ErrorMessage := '';
		16#802A:
			ErrorMessage := ' The header for the request is missing or invalid. ';
		16#802B:
			ErrorMessage := 'The timestamps to return parameter is invalid.';
		16#802C:
			ErrorMessage := 'The request was canceled by the client.';
//		16#802D:
//		ErrorMessage := '';
//		16#802E:
//		ErrorMessage := '';
//		16#802F:
//		ErrorMessage := '';

//		16#8030:
//		ErrorMessage := '';
		16#8031:
			ErrorMessage := 'Communication with the data source is defined but not established, and there is no last known value available.';
		16#8032:
			ErrorMessage := ' Waiting for the server to obtain values from the underlying data source. ';
		16#8033:
			ErrorMessage := 'The syntax of the node ID is not valid.';
		16#8034:
			ErrorMessage := 'The node ID refers to a node that does not exist in the server address space.';
		16#8035:
			ErrorMessage := 'The attribute is not supported for the specified node.';
		16#8036:
			ErrorMessage := 'The syntax of the index range parameter is invalid. ';
		16#8037:
			ErrorMessage := 'No data exists within the range of indexes specified.';
		16#8038:
			ErrorMessage := 'The data encoding is invalid.';
		16#8039:
			ErrorMessage := 'The server does not support the requested data encoding for the node.';
		16#803A:
			ErrorMessage := 'The access level does not allow reading or subscribing to the node.';
		16#803B:
			ErrorMessage := 'The access level does not allow writing to the node.';
		16#803C:
			ErrorMessage := 'The value was out of range.';
		16#803D:
			ErrorMessage := 'The requested operation is not supported.';
		16#803E:
			ErrorMessage := 'A requested item was not found or a search operation ended without success ';
		16#803F:
			ErrorMessage := 'The object cannot be used because it has been deleted.';

		16#8040:
			ErrorMessage := 'Requested operation is not implemented.';
		16#8041:
			ErrorMessage := 'The monitoring mode is invalid.';
		16#8042:
			ErrorMessage := 'The monitoring item ID does not refer to a valid monitored item.';
		16#8043:
			ErrorMessage := 'The monitored item filter parameter is not valid.';
		16#8044:
			ErrorMessage := 'The server does not support the requested monitored item filter.';
		16#8045:
			ErrorMessage := 'A monitoring filter cannot be used in combination with the attribute specified.';
		16#8046:
			ErrorMessage := 'A mandatory structured parameter was missing or null.';
		16#8047:
			ErrorMessage := 'The event filter is not valid.Identifier unknown';
		16#8048:
			ErrorMessage := 'The content filter is not valid.';
		16#8049:
			ErrorMessage := 'The operand used in a content filter is not valid.';
		16#804A:
			ErrorMessage := 'The continuation point provided is no longer valid.';
		16#804B:
			ErrorMessage := 'The operation could not be processed because all continuation points have been allocated.';
		16#804C:
			ErrorMessage := 'The reference type ID does not refer to a valid reference type node.';
		16#804D:
			ErrorMessage := 'The browse direction is not valid.';
		16#804E:
			ErrorMessage := 'The node is not part of the view.';
		16#804F:
			ErrorMessage := 'The server URI is not a valid URI.';

		16#8050:
			ErrorMessage := 'No server name was specified.';
		16#8051:
			ErrorMessage := 'No discovery URL was specified.';
		16#8052:
			ErrorMessage := 'The semaphore file specified by the client is not valid.';
		16#8053:
			ErrorMessage := 'The security token request type is not valid.';
		16#8054:
			ErrorMessage := 'The security mode does not meet the requirements set by the server.';
		16#8055:
			ErrorMessage := 'The security policy does not meet the requirements set by the server.';
		16#8056:
			ErrorMessage := 'The server has reached its maximum number of sessions.';
		16#8057:
			ErrorMessage := 'The user token signature is missing or invalid.';
		16#8058:
			ErrorMessage := 'The signature generated with the client certificate is missing or invalid.';
		16#8059:
			ErrorMessage := 'The client did not provide at least one software certificate that is valid and meets the profile requirements for the server.';
		16#805A:
			ErrorMessage := 'The request was canceled by the client with the cancel service.';
		16#805B:
			ErrorMessage := 'The parent node ID does not to refer to a valid node.';
		16#805C:
			ErrorMessage := 'The reference could not be created because it violates limitations imposed by the data model.';
		16#805D:
			ErrorMessage := 'The requested node ID was reject because it was either invalid or server does not allow node IDs to be specified by the client.';
		16#805E:
			ErrorMessage := 'The requested node ID is already used by another node.';
		16#805F:
			ErrorMessage := 'The node class is not valid.';

		16#8060:
		ErrorMessage := 'The browse name is invalid.';
		16#8061:
		ErrorMessage := 'The browse name is not unique among nodes that share the same relationship with the parent.';
		16#8062:
		ErrorMessage := 'The node attributes are not valid for the node class.';
		16#8063:
		ErrorMessage := 'The type definition node ID does not reference an appropriate type node.';
		16#8064:
		ErrorMessage := 'The source node ID does not reference a valid node. ';
		16#8065:
		ErrorMessage := 'The target node ID does not reference a valid node.';
		16#8066:
		ErrorMessage := 'The reference type between the nodes is already defined.';
		16#8067:
		ErrorMessage := 'The server does not allow this type of self reference on this node. ';
		16#8068:
		ErrorMessage := 'The reference type is not valid for a reference to a remote server. ';
		16#8069:
		ErrorMessage := 'The server will not allow the node to be deleted. ';
		16#806A:
		ErrorMessage := 'The server index is not valid. ';
		16#806B:
		ErrorMessage := 'The view ID does not refer to a valid view node.';
//		16#806C:
//		ErrorMessage := '';
		16#806D:
		ErrorMessage := 'The requested operation has too many matches to return.';
		16#806E:
		ErrorMessage := 'The requested operation requires too many resources in the server.';
		16#806F:
		ErrorMessage := 'The requested operation has no match to return.';

		16#8070:
		ErrorMessage := ' The max age parameter is invalid. ';
		16#8071:
		ErrorMessage := 'The history details parameter is not valid.';
		16#8072:
		ErrorMessage := 'The server does not support the requested operation.';
		16#8073:
		ErrorMessage := 'The server not does support writing the combination of value, status and timestamps provided.';
		16#8074:
		ErrorMessage := 'The value provided for the attribute is not of the same type as the attributes value.';
		16#8075:
		ErrorMessage := 'The method ID does not refer to a method for the specified object.';
		16#8076:
		ErrorMessage := 'The client did not specify all of the input arguments for the method. ';
		16#8077:
		ErrorMessage := 'The server has reached its maximum number of subscriptions.';
		16#8078:
		ErrorMessage := 'The server has reached the maximum number of queued publish requests.';
		16#8079:
		ErrorMessage := 'There is no subscription available for this session. ';
		16#807A:
		ErrorMessage := 'The sequence number is unknown to the server.';
		16#807B:
		ErrorMessage := 'The requested notification message is no longer available.';
		16#807C:
		ErrorMessage := 'The client of the current session does not support one or more profiles required for the subscription.';
		16#807D:
		ErrorMessage := 'The server cannot process the request because it is too busy.';
		16#807E:
		ErrorMessage := 'The type of the message specified in the header invalid.';
		16#807F:
		ErrorMessage := 'The secure channel ID and/or token ID are not currently in use.';

		16#8080:
			ErrorMessage := 'The size of the message specified in the header is too large.';
		16#8081:
			ErrorMessage := 'There are not enough resources to process the request.';
		16#8082:
			ErrorMessage := 'An internal error occurred.';
		16#8083:
			ErrorMessage := 'The server does not recognize the query string specified.';
		16#8084:
			ErrorMessage := 'The request could not be sent because of a network interruption.';
		16#8085:
			ErrorMessage := 'Timeout occurred while processing the request';
		16#8086:
			ErrorMessage := 'The secure channel has been closed.';
		16#8087:
			ErrorMessage := 'The token has expired or is not recognized.';
		16#8088:
			ErrorMessage := 'The sequence number is not valid.';
		16#8089:
			ErrorMessage := 'There is a problem with the configuration that affects the usefulness of the value';
		16#808A:
			ErrorMessage := 'The variable should receive its value from another variable, but has never been configured to do so.';
		16#808B:
			ErrorMessage := 'There has been a failure in the device/data source that generates the value that has affected the value.';
		16#808C:
			ErrorMessage := 'There has been a failure in the sensor from which the value is derived by the device/data source.';
		16#808D:
			ErrorMessage := 'The source of the data is not operational.';
		16#808E:
			ErrorMessage := 'The deadband filter is not valid.';
//		16#808F:
//		ErrorMessage := '';

//		16#8090:
//		ErrorMessage := '';
//		16#8091:
//		ErrorMessage := '';
//		16#8092:
//		ErrorMessage := '';
//		16#8093:
//		ErrorMessage := '';
//		16#8094:
//		ErrorMessage := '';
//		16#8095:
//		ErrorMessage := '';
//		16#8096:
//		ErrorMessage := '';
		16#8097:
			ErrorMessage := 'This condition refresh failed; a condition refresh operation is already in progress.';
		16#8098:
			ErrorMessage := 'This condition has already been disabled.';
		16#8099:
			ErrorMessage := ' Property not available, this condition is disabled. ';
		16#809A:
			ErrorMessage := 'The specified event ID is not recognized.';
		16#809B:
			ErrorMessage := ' No data is available for the desired time domain or event filter. ';
//		16#809C:
//		ErrorMessage := '';
		16#809D:
			ErrorMessage := 'Data is missing due to collection started/stopped/lost.';
		16#809E:
			ErrorMessage := 'Expected data is unavailable for the requested time range due to an unmounted data storage medium, an offline archive or tape or similar reason for temporary unavailability.';
		16#809F:
			ErrorMessage := ' The data or event was not successfully inserted because a matching entry exists.';

		16#80A0:
			ErrorMessage := 'The data or event was not successfully updated because no matching entry exists.';
		16#80A1:
			ErrorMessage := 'The client requested history using a timestamp format the server does not support (i.e requested server timestamp when server only supports source timestamp).';
//		16#80A2:
//		ErrorMessage := '';
//			16#80A3:
//		ErrorMessage := '';
//			16#80A4:
//		ErrorMessage := '';
//		16#80A5:
//		ErrorMessage := '';
//		16#80A6:
//		ErrorMessage := '';
//		16#80A7:
//		ErrorMessage := '';
//		16#80A8:
//		ErrorMessage := '';
//		16#80A9:
//		ErrorMessage := '';
//		16#80AA:
//		ErrorMessage := '';
		16#80AB:
			ErrorMessage := 'One or more arguments are invalid.';
		16#80AC:
			ErrorMessage := 'Could not establish a network connection to remote server.';
		16#80AD:
			ErrorMessage := 'The server has disconnected from the client.';
		16#80AE:
			ErrorMessage := 'The network connection has been closed.';
		16#80AF:
			ErrorMessage := 'The operation cannot be completed because the object is closed, uninitialized or in some other invalid state.';

		16#80B0:
		ErrorMessage := 'Cannot move beyond end of the stream.';
		16#80B1:
		ErrorMessage := 'No data is currently available for reading from a non-blocking stream.';
		16#80B2:
		ErrorMessage := 'The asynchronous operation is waiting for a response. ';
		16#80B3:
		ErrorMessage := 'The asynchronous operation was abandoned by the caller. ';
		16#80B4:
		ErrorMessage := 'The stream did not return all data requested (possibly because it is a non-blocking stream).';
		16#80B5:
		ErrorMessage := 'Non-blocking behavior is required and the operation would block.';
		16#80B6:
		ErrorMessage := 'A value had an invalid syntax.';
		16#80B7:
		ErrorMessage := 'The operation could not be finished because all available connections are in use.';
		16#80B8:
		ErrorMessage := 'The request message size exceeds limits set by the server.';
		16#80B9:
		ErrorMessage := 'The response message size exceeds limits set by the client.';
//		16#80BA:
//		ErrorMessage := '';
		16#80BB:
		ErrorMessage := ' The event cannot be acknowledged. ';
//		16#80BC:
//		ErrorMessage := '';
		16#80BD:
		ErrorMessage := 'The defined timestamp to return was invalid.';
		16#80BE:
		ErrorMessage := 'The applications do not have compatible protocol versions.';
		16#80BF:
		ErrorMessage := 'The sub-state machine is not currently active.';

//		16#80C0:
//		ErrorMessage := '';
		16#80C1:
		ErrorMessage := ' An unrecognized operator was provided in a filter. ';
		16#80C2:
		ErrorMessage := 'A valid operator was provided, but the server does not provide support for this filter operator.';
		16#80C3:
		ErrorMessage := 'The number of operands provided for the filter operator was less then expected for the operand provided.';
		16#80C4:
		ErrorMessage := 'The referenced element is not a valid element in the content filter.';
		16#80C5:
		ErrorMessage := 'The referenced literal is not a valid value.';
		16#80C6:
		ErrorMessage := 'The server does not support changing the user identity assigned to the session.';
//		16#80C7:
//		ErrorMessage := '';
		16#80C8:
		ErrorMessage := 'The provided node ID was not a type definition node ID. ';
		16#80C9:
		ErrorMessage := 'The view timestamp is not available or not supported.';
		16#80CA:
		ErrorMessage := 'The view parameters are not consistent with each other.';
		16#80CB:
		ErrorMessage := 'The view version is not available or not supported';
		16#80CC:
		ErrorMessage := 'This condition has already been enabled.';
		16#80CD:
		ErrorMessage := 'The dialog box state is not active.';
		16#80CE:
		ErrorMessage := 'The response is not valid for the dialog box.';
		16#80CF:
		ErrorMessage := ' The condition branch has already been acknowledged. ';

		16#80D0:
			ErrorMessage := 'The condition branch has already been confirmed.';
		16#80D1:
			ErrorMessage := 'The condition has already been shelved.';
		16#80D2:
			ErrorMessage := 'The condition is not currently shelved.';
		16#80D3:
			ErrorMessage := 'The shelving time not within an acceptable range.';
		16#80D4:
			ErrorMessage := 'The requested number of aggregates does not match the requested number of node IDs.';
		16#80D5:
			ErrorMessage := ' The requested aggregate is not support by the server.';
		16#80D6:
			ErrorMessage := 'The aggregate value could not be derived due to invalid data inputs.';
		16#80D7:
			ErrorMessage := 'No data found to provide upper or lower bound value.';
		16#80D8:
			ErrorMessage := 'The server cannot retrieve a bound for the variable.';
//		16#80D9:
//			ErrorMessage := '';
		16#80DA:
			ErrorMessage := 'The aggregate configuration is not valid for specified node.';
		16#80DB:
			ErrorMessage := ' The request could not be processed because there are too many monitored items in the subscription. ';
//		16#80DC:
//		ErrorMessage := '';
//		16#80DD:
//		ErrorMessage := '';
//		16#80DE:
//		ErrorMessage := '';
//		16#80DF:
//		ErrorMessage := '';

		ELSE
			ErrorMessage := '';
	END_CASE;

END_FUNCTION_BLOCK
```

### Types.typ
```iecst
TYPE
	csp_data_typ : 	STRUCT
		Customer : UDINT;
		Name : STRING[10];
		PermissionToLoad : BOOL;
	END_STRUCT;
	csp_typ : 	STRUCT
		Customer : UDINT;
		Data : ARRAY[0..1]OF csp_data_typ;
	END_STRUCT;
END_TYPE
```

### Variables.var
```iecst
VAR
	CSP : ARRAY[0..1] OF csp_typ;
	CurrentTimestamp : DATE_AND_TIME;
END_VAR
```

### Program Logical/CSP_Control/csp_control (IEC)

#### Main.st
```iecst
PROGRAM _INIT

END_PROGRAM

PROGRAM _CYCLIC

CSP[0].Customer;

END_PROGRAM

PROGRAM _EXIT
	(* Insert code here *)

END_PROGRAM
```

### Program Logical/CSP_Control/zzGetTime (IEC) - *Gets current timestamp

#### zzGetTimeCyclic.ab - Cyclic code
```automation-basic
(********************************************************************
 * COPYRIGHT -- HP
 ********************************************************************
 * Program: zzGetTime
 * File: zzGetTimeCyclic.ab
 * Author: treamsbottom
 * Created: June 04, 2014
 ********************************************************************
 * Implementation of program zzGetTime
 ********************************************************************)

PROGRAM _CYCLIC

	GetTimeStamp.enable = TRUE
	GetTimeStamp FUB DTGetTime()
	IF GetTimeStamp.status = ERR_OK THEN
		CurrentTimestamp = GetTimeStamp.DT1
	ENDIF
;	D32[78] = UDINT(CurrentTimestamp);
;
;	//Set the current time.
;	//DTSetTime(enable, DT1, status)
;	setTimeStamp.enable := (D32[79] > 0)
;	setTimeStamp.DT1 := DT(D32[79]); 	CAST D32 TO DT
;	setTimeStamp FUB DTSetTime()
;	IF (setTimeStamp.status =  ERR_OK) THEN
;		D32[79] = 0
;	ENDIF

END_PROGRAM
```

#### zzGetTime.var - Local variables
```iecst
(********************************************************************
 * COPYRIGHT -- HP
 ********************************************************************
 * Program: zzGetTime
 * File: zzGetTime.var
 * Author: treamsbottom
 * Created: June 04, 2014
 ********************************************************************
 * Local variables of program zzGetTime
 ********************************************************************)
VAR
	GetTimeStamp : DTGetTime;
	setTimeStamp : DTSetTime;
END_VAR
```

### Request_Constants.var
```iecst
VAR CONSTANT
	HTTP_IF_CALL_USP_NOREPLY_URL : STRING[100] := '/httpcomms/api/plcToSql/calluspnoquery'; (**POST Put Procedure string in the body data*)
	HTTP_IF_CALL_USP_REPLY_URL : STRING[100] := '/httpcomms/api/plcToSql/callusp?sql='; (**GET Function - Put Procedure in URL*)
END_VAR
(*POST - USPS*)
VAR CONSTANT
	HTTP_POST_MAINT_COMPLETE : STRING[100] := '[SUPDB].[Maintenance].[uspMaintenanceBagMaintComplete]'; (*Maint Complete. Needs @PLC,@Bag*)
	HTTP_USP_WRITE_SEQ_COUNT_DATA : STRING[100] := '[SUPDB].[PLC].[uspWriteSequenceCount]'; (*Stored procedure uspWriteSequenceCount. Requires @PLCStn, @SeqNum, @CountIn*)
	HTTP_USP_WRITE_REPORT_DATA : STRING[100] := '[SUPDB].[PLC].[uspReportWrite]'; (*Stored procedure uspReportWrite*)
	HTTP_POST_BATCH_LOCATION_UPDATE : STRING[100] := '[SUPDB].[Master].[uspBatch_LocationUpdate]'; (*Stored procedure [Master].[uspBatch_LocationUpdate] Update batch location.
*)
	HTTP_POST_BATCH_PROPERTY_UPDATE : STRING[100] := '[SUPDB].[Master].[uspBatch_Property_Update]'; (*Stored procedure [Master].[uspBatch_Property_Update] Update a single batch propery by name...
*)
END_VAR
(*GET*)
VAR CONSTANT
	HTTP_GET_SUPERTRACK_CON_STATUS : STRING[100] := '/supertrack/api/settings/connectOpc';
	HTTP_GET_OPCUA_CONNECTION_STATUS : STRING[100] := '/KanDisplay.Manager.API/api/settings/connectOpc';
	HTTP_GET_MAINT_COMPLETE : STRING[100] := '[SUPDB].[Maintenance].[uspMaintenanceBagMaintComplete]'; (*Maint Complete. Needs @PLC,@Bag*)
	HTTP_GET_MAINT_COUNT_REPLY_STATE : STRING[100] := '/maintenance.api/api/Bags/bagCountUpdate?bagNumber='; (*Send count value, reply state. Needs @PLC,@Bag, @State OUTPUT>.*)
	HTTP_GET_BATCH_CREATE_LOC_UPDATE : STRING[100] := '[SUPDB].[Master].[uspBatch_Create_UpdateLocation]'; (*Update batch location, or create batch if it doesn't exist.*)
END_VAR
(*MIS Batch Interface ADRETT SPECIAL*)
VAR CONSTANT
	HTTP_GET_BATCH_CREATE : STRING[100] := '[SUPDB].[PLC].[uspMIS_BatchCreate]'; (*Update batch location, or create batch if it doesn't exist.*)
END_VAR
```

### Server_Functions.var
```iecst
VAR CONSTANT
	HTTP_SVR_FNC_NOT_FOUND : UINT := 0;
	HTTP_SVR_GET_FNC_RESTART_PLC : UINT := 4;
	HTTP_SVR_GET_FNC_SET_BAG_DEST : UINT := 1;
	HTTP_SVR_GET_FNC_TEST : UINT := 2;
	HTTP_SVR_POST_FNC_TEST : UINT := 20;
END_VAR
```

### Constants.var
```iecst
VAR CONSTANT
	STRING_DOLLAR : STRING[1] := '&';
	STRING_COMMA : STRING[1] := ',';
END_VAR
```

### Variables.var
```iecst
VAR CONSTANT
	HTTP_MAX_COMM : UINT := 20; (**Max number of interfaces to talk to http.*)
END_VAR
VAR
	HTTP_Comm : ARRAY[0..HTTP_MAX_COMM] OF http_comm_typ;
	HTTP_Config : httpConfig_typ;
END_VAR
VAR CONSTANT
	DEFAULT_REQUEST_HEADER : httpRequestHeader_t := (protocol:='HTTP/1.1',host:='10.8.4.220',contentType:='text/plain',connection:='keep-alive',keepAlive:='max=100,timeout=10');
END_VAR
```

### Types.typ - Exported data types
```iecst
TYPE
	dataPointer_typ : 	STRUCT
		Adr : UDINT;
		Size : UDINT;
	END_STRUCT;
	httpConfig_typ : 	STRUCT
		Host : STRING[20];
		Port : UINT;
	END_STRUCT;
	http_Cmd_typ : 	STRUCT
		Method : UINT; (*Set the http cmd type.. POST,GET,PUT,DELETE*)
		Cmd_URL : dataPointer_typ; (*The string data appended to the URL - Use with GET and DELETE *)
		Body_Data : dataPointer_typ; (*Data to send in the body of the message - USE with POST and PUT*)
		ResponseData : dataPointer_typ; (*Data address of where to set the http response data*)
	END_STRUCT;
	http_comm_typ : 	STRUCT
		Command : http_Cmd_typ; (**Set the values to pass into the http comm driver,*)
		Status : HTTP_Status_enum; (**Status of the http comm driver.*)
		LastError : STRING[60]; (**String to describe the last error*)
		lastResponse : httpResponseHeader_t;
		Overwrite : http_overwrite_t;
		ReplyCode : UINT; (**The response code *)
	END_STRUCT;
	http_overwrite_t : 	STRUCT
		Host : BOOL; (**Set this to overwrite the host name and Port*)
		RequestHeader : BOOL; (**Set this to overwrite the Request Header*)
		Host_Config : httpConfig_typ; (**This data will overwrite the default host config*)
		RequestHeader_Data : httpRequestHeader_t; (**This data will overwrite the default request header.*)
	END_STRUCT;
	HTTP_Status_enum :
		(
		HTTP_COMM_STATUS_DISABLED,
		HTTP_COMM_STATUS_ACTIVE_WAIT_BUF,
		HTTP_COMM_STATUS_IN_BUFFER,
		HTTP_COMM_STATUS_IN_PROCESS,
		HTTP_COMM_STATUS_COMPLETE,
		HTTP_COMM_STATUS_ERROR
		);
END_TYPE

(*Response Data from LiveData*)
```

- Http_Info.docx (binary file, 16280 bytes)
### Library Logical/http_Lib/KanHttp (IEC)
Depends on: AsHttp, AsFifo

#### Constants.var - Exported constants
```iecst
VAR CONSTANT
	API_UNKNOWN : USINT := 0;
	API_MAINTENANCE_CONFIRM_REENTRY : USINT := 1;
	API_DISCHARGER_SUBMIT : USINT := 3;
	API_LOADING_NEWDATA : USINT := 4;
	API_LOADING_SUBMIT : USINT := 5;
	API_LOADING_WITH_TOUR_NEWDATA : USINT := 10;
	API_LOADING_WITH_TOUR_SUBMIT : USINT := 11;
	API_CUSTOMER_CHANGE : USINT := 20;
	API_ABB_MANUAL_CMD : USINT := 30;
	API_NEDLIN_GET_CSP_DATA : USINT := 40;
	API_NEDLIN_SET_CSP_DATA : USINT := 41;
	API_RESET_SORTING_COUNT : USINT := 50;
	API_UPDATE_VAR_BY_NAME : USINT := 90;
	API_CONFIG_LOAD_NEW : USINT := 91;
	API_CONFIG_SAVE : USINT := 92;
	API_ST_FUNCTIONS : USINT := 99;
END_VAR
```

#### KanHttp.fun - Exported functions and function blocks
```iecst
FUNCTION_BLOCK httpGetParameter (*FUB to Get parameter values set in URI or BODY...*) (*$GROUP=User,$CAT=User,$GROUPICON=User.png,$CATICON=User.png*)
	VAR_INPUT
		searchPropertyName : STRING[50]; (*StringValue of propery or name to match*)
		searchEndProperty : STRING[50]; (*String Character or value to show end of property value -- DEFAULT & *)
		searchOffset : UINT; (*Offset can be set to skip searching begining of string if not required*)
		searchString : {REDUND_UNREPLICABLE} STRING[5000];
	END_VAR
	VAR_OUTPUT
		outputValue : STRING[100]; (*String Value found*)
		status : UINT;
		postionFound : UINT; (*Start position of the data found *)
	END_VAR
	VAR
		matchString : STRING[50];
		inputData : ARRAY[0..4999] OF USINT;
		endIndex : UINT;
		startPosition : UINT;
		n : UINT;
		compare : DINT;
		length : UINT;
		startoffset : UINT;
		search : STRING[50];
	END_VAR
END_FUNCTION_BLOCK

FUNCTION FindAPI : UINT (**Get API name from URI*) (*$GROUP=User,$CAT=User,$GROUPICON=User.png,$CATICON=User.png*)
	VAR_INPUT
		URI : STRING[500];
		ServiceName : STRING[50];
	END_VAR
	VAR
		Length : INT;
		Start : INT;
		apiName : STRING[100];
	END_VAR
END_FUNCTION
```

#### httpGetParameter.st
```iecst
(* FUB to Get parameter values set in URI or BODY... *)
FUNCTION_BLOCK httpGetParameter
	status := ERR_FUB_BUSY;
// Get the function Name from the URI
//Use the string length of the service name	+
	memset(ADR(outputValue),0,SIZEOF(outputValue));
	matchString := searchPropertyName;
	strcpy(ADR(inputData[0]),ADR(searchString));
	startoffset := searchOffset;
	endIndex := LEN(searchString);
	startPosition := 16#FFF;
	IF endIndex > startoffset THEN
		FOR n := startoffset TO endIndex DO
			memcpy(ADR(search),ADR(inputData[n]),LEN(matchString));
			compare := 	strcmp(ADR(search),ADR(matchString));
			IF (compare = 0) THEN
				startPosition := n + LEN(matchString);
				EXIT;
			END_IF;
		END_FOR;
	ELSE
		status := 100;
	END_IF;

	IF (startPosition <> 16#FFF) THEN
		//Get the End Position
		matchString := searchEndProperty;
		memset(ADR(search),0,SIZEOF(search));
		startoffset := startPosition;
		IF endIndex >= startoffset THEN
			FOR n := startoffset TO endIndex DO
				memcpy(ADR(search),ADR(inputData[n]),LEN(matchString));
				compare := 	strcmp(ADR(search),ADR(matchString));
				length := n - startPosition;
				IF (compare = 0) THEN
					EXIT;
				END_IF;
			END_FOR;
			outputValue := MID(searchString,length,startPosition + 1);
			postionFound := n;
			status := ERR_OK;
		ELSE
			status := 102;
		END_IF;
	ELSE
		outputValue := '';
		status := 101;
	END_IF;

END_FUNCTION_BLOCK
```

#### FindAPI.st
```iecst
(* *Get API name from URI *)
FUNCTION FindAPI

	Start := LEN(ServiceName) + 2;// We must add the / character and 1 to place the cursor on the first Letter of the API name.
	Length := FIND(URI,'?');
	IF (Length = 0) THEN
		Length := LEN(URI)- LEN(ServiceName) + 1;;
	ELSE
		Length := Length - LEN(ServiceName) - 2;
	END_IF;

	apiName := 	MID(URI,Length,Start);

	IF (apiName = 'ConfirmBagReEntry') THEN FindAPI := API_MAINTENANCE_CONFIRM_REENTRY;
	ELSIF (apiName = 'Functions') THEN FindAPI := API_ST_FUNCTIONS;
//	ELSIF (apiName = 'SendBeltLoadingConfig') THEN FindAPI := API_CUSTOM_BELT_CONFIG;

	ELSIF (apiName = 'discharger-submit') THEN FindAPI := API_DISCHARGER_SUBMIT;
	ELSIF (apiName = 'abb-manual-control') THEN FindAPI := API_ABB_MANUAL_CMD;
	ELSIF (apiName = 'submit-customer-change') THEN FindAPI := API_CUSTOMER_CHANGE;
	ELSIF (apiName = 'loading-screen-submit') THEN FindAPI := API_LOADING_SUBMIT;
	ELSIF (apiName = 'loading-screen-changed') THEN FindAPI := API_LOADING_NEWDATA;
	ELSIF (apiName = 'loading-screen-with-tour-submit') THEN FindAPI := API_LOADING_WITH_TOUR_SUBMIT;
	ELSIF (apiName = 'loading-screen-with-tour-changed') THEN FindAPI := API_LOADING_WITH_TOUR_NEWDATA;
	ELSIF (apiName = 'update-var-by-name') THEN FindAPI := API_UPDATE_VAR_BY_NAME;
	ELSIF (apiName = 'commit-updates') THEN FindAPI := API_CONFIG_SAVE;
	ELSIF (apiName = 'load-config') THEN FindAPI := API_CONFIG_LOAD_NEW;
	ELSIF (apiName = 'nedlin-get-csp-data') THEN FindAPI := API_NEDLIN_GET_CSP_DATA;
	ELSIF (apiName = 'nedlin-set-csp-data') THEN FindAPI := API_NEDLIN_SET_CSP_DATA;
	ELSIF (apiName = 'reset-sorting-count') THEN FindAPI := API_RESET_SORTING_COUNT;
	ELSE FindAPI := API_UNKNOWN;
	END_IF;

END_FUNCTION
```

### Program Logical/http_Lib/httpServer (IEC, version 9.99.9) - *Listen for http requests

#### Variables.var - Local variables
```iecst
VAR
	httpServer : httpService;
	sendResponse : BOOL;
	abortResponse : BOOL;
	URI : STRING[500];
	requestHeader : httpRequestHeader_t;
	requestData : STRING[10000];
	responseHeader : httpResponseHeader_t;
	responseData : STRING[10000];
	Statistics : httpStatistics_t;
	serviceName : STRING[50];
	getParameterName : httpGetParameter;
END_VAR
VAR CONSTANT
	STRING_DOLLAR : STRING[1] := '&';
END_VAR
VAR
	activeFunction : UINT;
	mis : UDINT;
	bagIndex : UDINT;
	dst : USINT;
	error : INT;
	api : UINT;
	errorResponse : BOOL;
	overRideData : overRide_typ;
	ton_httpTimeOut : TON_10ms;
	recv : R_TRIG;
	wait : F_TRIG;
	cat : UDINT;
	cus : UDINT;
	prg : USINT;
	found : USINT;
	recieved : BOOL;
END_VAR
VAR CONSTANT
	BLANK_RESPONSE_HEADER : httpResponseHeader_t := (0);
END_VAR
VAR
	requestArriveTime : DATE_AND_TIME;
	debugCount : UDINT;
	index : UDINT;
	belt : USINT;
	velocity : INT;
	direction : USINT;
	command : USINT;
	sp1 : UINT;
	sp2 : UINT;
	sp3 : UINT;
	tourID : UDINT;
	varName : STRING[100];
	setValue : USINT;
	status : UINT;
	pv_adr : UDINT;
	pv_len : UDINT;
	value : STRING[100];
	pv_type : UDINT;
	pv_length : UDINT;
	pv_dimension : UINT;
	isString : BOOL;
	stringCheck : BOOL;
	num_Val : DINT;
	float_val : REAL;
	clearFifo : fifoClear;
	createFifo : fifoCreate;
	deleteFifo : fifoDelete;
	scanCount : USINT;
	searchOffset : UINT;
END_VAR
VAR CONSTANT
	SEARCH_STRING_VAR_NAME : STRING[20] := 'varName":"';
	SEARCH_STRING_VAR_VALUE : STRING[20] := 'value":';
END_VAR
VAR
	writeFifo : fifoWrite;
	arrayEnd : UINT;
	data : ARRAY[0..1] OF UDINT;
	fi_status : UDINT;
	pData : UDINT;
	pos1 : UINT;
	pos2 : UINT;
	readFifo : fifoRead;
	string_Val : STRING[100];
	length : UDINT;
	responseDataBinary : ARRAY[0..1999] OF USINT;
	sendBinaryData : BOOL;
END_VAR
```

#### Main.st - Init, cyclic, exit code
```iecst
//V2.00.1 -- TR. First release using version numbering
//V2.00.2 -- TR. Remove old http server functions FOR ABB settings as vars have been removed
//		  -- FIX: 200 OK could be returned in error
//V2.00.3 -- ADD: Load new configuration file command
//V2.00.4 -- REMOVE: Clear up old API Calls
//V2.00.5 -- Add Discharger Displays
//V2.00.6 -- ADD Part load and ABB Manual Controls (NEEDS ABB DRIVER 3.00.2)
//V2.00.7 -- ADD more functionality to ABB Manual Controls (Command and Direction)
//V3.00.1 -- Standardise the response data from LiveData displays
//V3.00.2 -- ADD Update var by name endpoint
//V3.00.3 -- FIX - Range issues in updateVarByName - ADD HTTP CALLS FOR PLC-CONFIG.Web

//V9.99.9  -- Special version for NEDLIN

PROGRAM _INIT
	serviceName := 'supertrackPLC.api';
	httpServer.pServiceName := ADR(serviceName);
	httpServer.pUri := ADR(URI);
	httpServer.uriSize := SIZEOF(URI);
	httpServer.pRequestHeader := ADR(requestHeader);
	httpServer.pRequestData := ADR(requestData);
	httpServer.requestDataSize := SIZEOF(requestData);
	httpServer.pResponseHeader := ADR(responseHeader);

	httpServer.pStatistics := ADR(Statistics);

	httpServer.option := httpOPTION_HTTP_11 + httpOPTION_SERVICE_TYPE_ROOT; //HTTP 1.1
	httpServer.enable := 0;

END_PROGRAM

PROGRAM _CYCLIC

	_httpServer;

	wait(CLK := (httpServer.phase = httpPHASE_SENDING));
	recv(CLK := (httpServer.phase = httpPHASE_RECEIVED));
	IF wait.Q THEN
		memset(ADR(responseData),0,SIZEOF(responseData));//Clear responseData
		memset(ADR(responseDataBinary),0,SIZEOF(responseDataBinary));
		found	:= 0;
		error := 0;
	END_IF;

	IF EDGEPOS(recieved) THEN
		requestArriveTime := CurrentTimestamp; // Get time stamp when the request arrives.
	END_IF;

	IF recieved THEN//recv.Q THEN
		//Get the API!
		api := FindAPI(URI,serviceName);

		CASE api OF

			API_UNKNOWN:
				errorResponse := 1;
				overRideData.responseHeader.status := '501 Not Implemented';
				responseData := 'Unknown API';
				httpServer.responseDataLen := LEN(responseData);

//			API_MAINTENANCE_CONFIRM_REENTRY:
//				sendResponse := 1;

			API_ST_FUNCTIONS://Legacy function => ?function=xxx
				_apiFunctions;

//			API_DISCHARGER_SUBMIT:
//
//				getParameterName.searchString := requestData;
//				getParameterName.searchOffset := 0;
//				getParameterName.searchEndProperty := STRING_DOLLAR;
//				//Find the first part of the array in JSON
//				getParameterName.searchPropertyName := 'playId":"';
//				getParameterName.searchEndProperty := '",';
//				getParameterName();
//				IF (getParameterName.status = ERR_OK) THEN
//					index := DINT_TO_UDINT(atoi(ADR(getParameterName.outputValue)));
//					IF (index <= MAX_DISPLAYS) THEN
//						LiveData_Recv[index].Submit_Discharger := 1;
//					END_IF;
//					sendResponse := 1;
//				ELSE
//					errorResponse := 1;
//					overRideData.responseHeader.status := '404 Not Found';
//					responseData := 'Unknown display';
//					httpServer.responseDataLen := LEN(responseData);
//				END_IF;

//			API_ABB_MANUAL_CMD:
//				_abbManual;
//
//			API_CUSTOMER_CHANGE:
//				_customerChange;
//
//			API_LOADING_SUBMIT:
//				_getLoadingSubmit;
//
//			API_LOADING_NEWDATA:
//				_getLoadingData;
//
//			API_LOADING_WITH_TOUR_SUBMIT:
//				_getTourLoadingSubmit;
//
//			API_LOADING_WITH_TOUR_NEWDATA:
//				_getTourLoadingData;
//
//			API_UPDATE_VAR_BY_NAME:
//				_updateVarByName;
//
//			API_CONFIG_LOAD_NEW: // Request to load new configuration.
//				IF (Configuration.Interface.Status.LastLoaded >= requestArriveTime)  THEN // Send 200 OK when we see that the configuration is newer than the previous
//					sendResponse := 1;
//				ELSIF Configuration.Interface.Status.Error THEN
//					errorResponse := 1;
//					overRideData.responseHeader.status := '500 Internal Server Error';
//					responseData := 'Failed to load file';
//					httpServer.responseDataLen := LEN(responseData);
//				ELSIF NOT Configuration.Interface.Cmd.Load AND (Configuration.Interface.Status.LastLoaded < requestArriveTime) THEN
//					Configuration.Interface.Cmd.Load := 1;
//					debugCount := debugCount + 1;
//				END_IF;
//
//			API_CONFIG_SAVE:
//
//				IF (Configuration.Interface.Status.LastSaved >= requestArriveTime)  THEN // Send 200 OK when we see that the configuration is newer than the previous
//					sendResponse := 1;
//				ELSIF Configuration.Interface.Status.Error THEN
//					errorResponse := 1;
//					overRideData.responseHeader.status := '500 Internal Server Error';
//					responseData := 'Failed to save file';
//					httpServer.responseDataLen := LEN(responseData);
//				ELSIF NOT Configuration.Interface.Cmd.Save AND (Configuration.Interface.Status.LastSaved < requestArriveTime) THEN
//					Configuration.Interface.Cmd.Save := 1;
//				END_IF;

			API_NEDLIN_GET_CSP_DATA: // Get the current CSP data status.
				length := SIZEOF(CSP);
				overRideData.responseHeader.contentType := 'nothing';
				brsmemcpy(ADR(responseDataBinary),ADR(CSP),length);
				overRideData.responseDataLen := length;
				sendResponse := 1;
				sendBinaryData := 1;

			API_NEDLIN_SET_CSP_DATA: //  Set the incoming customers
				_nedlinSetCustomer;

			API_RESET_SORTING_COUNT:
				_resetCount;

		END_CASE;
	ELSE
		api := 0;
		activeFunction := 0;
	END_IF;

END_PROGRAM

PROGRAM _EXIT
	//Disable the Server on Exit..
	httpServer.enable := 0;
	httpServer();
END_PROGRAM
```

#### _vcCommand.st
```iecst
ACTION _vcCommand:
	//IF VC_Command[1] = VC_CMD_NOTHING THEN
		getParameterName.searchString := requestData;
		getParameterName.searchPropertyName := 'command":"';
		getParameterName.searchEndProperty := '"';
		getParameterName.searchOffset := 0;
		getParameterName();
		IF (getParameterName.status = ERR_OK) THEN
			IF getParameterName.outputValue = 'get-empty-bag' THEN
				VC_Command[1] := VC_CMD_GOTO_EMPTY;
			ELSIF getParameterName.outputValue = 'bag-removed' THEN
				VC_Command[1] := VC_CMD_BAG_REMOVED_CONFIRM;
			ELSIF getParameterName.outputValue = 'load-maintenance-bag' THEN
				VC_Command[1] := VC_CMD_LOAD_MAINT_BAG;
			ELSIF getParameterName.outputValue = 'go-to-loading' THEN
				VC_Command[1] := VC_CMD_GOTO_LOADING;
			ELSE
				errorResponse 	:= 1;
			END_IF;
		ELSE
			errorResponse := 1;
		END_IF;
//WE NEED TO HAVE A COMMAND RESPONSE SO WE CAN SEND THE CORRECT RESPONSE TO THE DISPLAY>>>

//	ELSE
//		IF (D[903] = 8) THEN
			sendResponse := 1;
//		ELSIF VC_Command[1] = VC_CMD_FAIL THEN
//			sendResponse := 1;
//			overRideData.responseHeader.status := '409 Conflict';
//		END_IF;
//	END_IF;
END_ACTION
```

#### _apiFunctions.st
```iecst
ACTION _apiFunctions:
	IF activeFunction = 0 THEN _getFunctionName; END_IF;
	//Exectute the Function
	CASE activeFunction OF
		HTTP_SVR_FNC_NOT_FOUND: //Nothing
			sendResponse := 1;
			memset(ADR(responseData),0,SIZEOF(responseData));//Clear responseData
			responseData := 'error Function Not found, Function Must be specified with function=';
			httpServer.responseDataLen := LEN(responseData);

		HTTP_SVR_GET_FNC_SET_BAG_DEST: //Set Bag Destination -- 1
		//				_setBagDestination;
		HTTP_SVR_GET_FNC_TEST://Test
			sendResponse := 1;
			memset(ADR(responseData),0,SIZEOF(responseData));//Clear responseData
			responseData := 'Test Get';
			httpServer.responseDataLen := LEN(responseData);

		HTTP_SVR_POST_FNC_TEST:
			//sendResponse := 1;
			memset(ADR(responseData),0,SIZEOF(responseData));//Clear responseData
			responseData := 'Test Post';
			httpServer.responseDataLen := LEN(responseData);

		HTTP_SVR_GET_FNC_RESTART_PLC:
			sendResponse := 1;
			memset(ADR(responseData),0,SIZEOF(responseData));//Clear responseData
			responseData := 'PLC will carry out a warm restart';
			httpServer.responseDataLen := LEN(responseData);
			IF httpServer.phase = 4 THEN //Wait for response to be sent
				SYSreset(TRUE,1); //Restart PLC
			END_IF;

	END_CASE

END_ACTION
```

#### _getFunctionName.st
```iecst
ACTION _getFunctionName:
	CASE httpServer.method OF
		httpMETHOD_DELETE,httpMETHOD_PUT:
			//wrong method-- implement error handling.

		httpMETHOD_GET:
			getParameterName.searchString := URI;
			getParameterName.searchOffset := LEN(serviceName);
		httpMETHOD_POST:
			getParameterName.searchString := URI;
			getParameterName.searchOffset := LEN(serviceName);
//			getParameterName.searchString := requestData;
//			getParameterName.searchOffset := 0;
	END_CASE;

	getParameterName.searchPropertyName := 'function=';
	getParameterName.searchEndProperty := STRING_DOLLAR ;
	getParameterName();

	CASE httpServer.method OF
		httpMETHOD_DELETE,httpMETHOD_PUT:
			//wrong method-- implement error handling.

		httpMETHOD_GET:
			IF getParameterName.status = ERR_OK THEN
				IF getParameterName.outputValue = 'dmSetDst' THEN activeFunction := HTTP_SVR_GET_FNC_SET_BAG_DEST;
				ELSIF getParameterName.outputValue = 'test' THEN activeFunction := HTTP_SVR_GET_FNC_TEST;
				ELSIF getParameterName.outputValue = 'restart' THEN activeFunction := HTTP_SVR_GET_FNC_RESTART_PLC;
				ELSE activeFunction := HTTP_SVR_FNC_NOT_FOUND;
				END_IF;
				getParameterName.searchString := '';
			END_IF;
		httpMETHOD_POST:
			IF getParameterName.status = ERR_OK THEN
				IF getParameterName.outputValue = 'test' THEN activeFunction := HTTP_SVR_POST_FNC_TEST;
				ELSE activeFunction := HTTP_SVR_FNC_NOT_FOUND;
				END_IF;
				getParameterName.searchString := '';
			END_IF;
	END_CASE;

END_ACTION
```

#### _setBagDestination.st
```iecst
ACTION _setBagDestination:

	mis := 0;
	bagIndex := 0;
	dst := 0;
	error := 0;

	//Set common parameters of the function.
	getParameterName.searchString := requestData;
	getParameterName.searchOffset := 0;
	getParameterName.searchEndProperty := STRING_DOLLAR ;

	//Get Mis Parameter
	getParameterName.searchPropertyName := 'mis=';
	getParameterName();
	IF getParameterName.status = ERR_OK THEN
		mis := DINT_TO_UDINT(atoi(ADR(getParameterName.outputValue)));
	ELSE
		error := 1;
	END_IF;

	//Get bag index Parameter
	getParameterName.searchPropertyName := 'bagindex=';
	getParameterName();
	IF getParameterName.status = ERR_OK THEN
		bagIndex := DINT_TO_UDINT(atoi(ADR(getParameterName.outputValue)));
	ELSE
		error := 2;
	END_IF;

	//Get Destination
	getParameterName.searchPropertyName := 'dest=';
	getParameterName();
	IF getParameterName.status = ERR_OK THEN
		dst := DINT_TO_USINT(atoi(ADR(getParameterName.outputValue)));
	ELSE
		error := 3;
	END_IF;

	CASE error OF
		0:// No Errors SEND //Check bag is correct.
			IF (bagIndex <= MAX_BAGS) THEN
				IF Bag[bagIndex].Cat > 0 THEN
					IF Bag[bagIndex].Mis = mis THEN
						IF dst <= MAX_LINES THEN
							Bag[bagIndex].Dst := dst;
							responseData := getParameterName.outputValue;
						ELSE
							responseData := 'error bag destination out of range';
						END_IF;
					ELSE
						responseData := 'error bag index and mis don;t match';
					END_IF;
				ELSE
					responseData := 'error bag at bag index is not valid - No Category';
				END_IF;
			ELSE
				responseData := 'error Bag index greater then bags';
			END_IF;
		1: //Mis Param not found
			responseData := 'error mis parameter not found';
		2: //bagindex Param not found
			responseData := 'error bagindex parameter not found';
		3: //Dest Param not found
			responseData := 'error dest parameter not found';
	END_CASE;

	sendResponse := 1;
	httpServer.responseDataLen := LEN(responseData);

END_ACTION
```

#### _setBeltConfig.st
```iecst
ACTION _setBeltConfig:

	bagIndex := 0;
	prg	:= 0;
	cat := 0;
	cus := 0;
	dst := 0;
	error := 0;
	found := 0;
	//Set common parameters of the function.
	getParameterName.searchString := requestData;
	getParameterName.searchOffset := 0;
	getParameterName.searchEndProperty := STRING_DOLLAR;
	REPEAT

		//Find the first part of the array in JSON
		getParameterName.searchPropertyName := '{';
		getParameterName.searchEndProperty := '"';
		getParameterName();
		IF (getParameterName.status = ERR_OK) THEN
			getParameterName.searchOffset := DINT_TO_UINT(getParameterName.nextPosition);
		ELSE
			error := 1;
		END_IF;

		//Find the category
		getParameterName.searchPropertyName := '"category":';
		getParameterName.searchEndProperty := ',';
		getParameterName();
		IF getParameterName.status = ERR_OK THEN
			cat := DINT_TO_UDINT(atoi(ADR(getParameterName.outputValue)));
		ELSE
			error := 2;
		END_IF;

		//Find the customer
		getParameterName.searchPropertyName := ',"customer":';
		getParameterName.searchEndProperty := ',';
		getParameterName();
		IF getParameterName.status = ERR_OK THEN
			cus := DINT_TO_UDINT(atoi(ADR(getParameterName.outputValue)));
		ELSE
			error := 2;
		END_IF;

		//Find the program
		getParameterName.searchPropertyName := '"program":';
		getParameterName.searchEndProperty := '}';
		getParameterName();
		IF getParameterName.status = ERR_OK THEN
			prg := DINT_TO_USINT(atoi(ADR(getParameterName.outputValue)));
			CASE found OF
				0:
					bag ACCESS ADR(Bag[340]);
				1:
					bag ACCESS ADR(Bag[364]);
				2:
					bag ACCESS ADR(Bag[350]);
			END_CASE;
			IF (found >= 0) AND (found <= 2) THEN
				found := found + 1;
				bag.Cat := cat;
				bag.Prg := prg;
				bag.Cus := cus;
				bag.Dst := dst;
			ELSE
				error := 7;
			END_IF;
		ELSE
			error := 3;
		END_IF;

	UNTIL ((error > 0) OR (found > 2))
	END_REPEAT;

	sendResponse := (found > 0);
	errorResponse := (error > 0);

END_ACTION
```

#### _customerChange.st
```iecst
ACTION _customerChange:
	//{"stationId":1,"cus":25,"plcStation":0}
	index := 0;
	cus := 0;

	error := 0;
	found := 0;
	//Set common parameters of the function.
	getParameterName.searchString := requestData;
	getParameterName.searchOffset := 0;
	getParameterName.searchEndProperty := STRING_DOLLAR;

	//Find the Index
	getParameterName.searchPropertyName := '"stationId":';
	getParameterName.searchEndProperty := ',';
	getParameterName();
	IF getParameterName.status = ERR_OK THEN
		index := DINT_TO_UDINT(atoi(ADR(getParameterName.outputValue)));
	ELSE
		error := 2;
	END_IF;

	//Find the customer
	getParameterName.searchPropertyName := '"cus":';
	getParameterName.searchEndProperty := ',';
	getParameterName();
	IF getParameterName.status = ERR_OK THEN
		cus := DINT_TO_USINT(atoi(ADR(getParameterName.outputValue)));
		IF (index <= MAX_DISPLAYS) THEN
			LiveData_Recv[index].Bag.Cus := cus;
			LiveData_Recv[index].Submit_CustomerChange := 1;
			found := found + 1;
		ELSE
			error := 99;
			overRideData.responseHeader.status := '404 Not Found';
			responseData := 'Unknown display';
			httpServer.responseDataLen := LEN(responseData);
		END_IF;
	ELSE
		error := 3;
	END_IF;

	sendResponse := (found > 0);
	errorResponse := (error > 0);

END_ACTION
```

#### _PostAbbManual.st
```iecst
ACTION _abbManual:
	//'{"belt":1,"speed":25,"direction":0,"command":1}'
	belt 		:= 0;
	velocity 	:= 0;
	direction 	:= 0;
	command 	:= 0;

	error := 0;
	found := 0;
	//Set common parameters of the function.
	getParameterName.searchString := requestData;
	getParameterName.searchOffset := 0;
	getParameterName.searchEndProperty := STRING_DOLLAR;

	//Find the id
	getParameterName.searchPropertyName := '"belt":';
	getParameterName.searchEndProperty := ',';
	getParameterName();
	IF getParameterName.status = ERR_OK THEN
		belt := DINT_TO_USINT(atoi(ADR(getParameterName.outputValue)));
		getParameterName.searchOffset := getParameterName.nextPosition;
	ELSE
		error := 1;
	END_IF;

	//set the velocity
	getParameterName.searchPropertyName := '"speed":';
	getParameterName.searchEndProperty := ',';
	getParameterName();
	IF getParameterName.status = ERR_OK THEN
		velocity := DINT_TO_INT(atoi(ADR(getParameterName.outputValue)));
	ELSE
		error := 2;
	END_IF;

	//set the direction
	getParameterName.searchPropertyName := '"direction":';
	getParameterName.searchEndProperty := ',';
	getParameterName();
	IF getParameterName.status = ERR_OK THEN
		direction := DINT_TO_USINT(atoi(ADR(getParameterName.outputValue)));
	ELSE
		error := 3;
	END_IF;

	getParameterName.searchPropertyName := '"command":';
	getParameterName.searchEndProperty := '}';
	getParameterName();
	IF getParameterName.status = ERR_OK THEN
		command := DINT_TO_USINT(atoi(ADR(getParameterName.outputValue)));
		IF (belt <= MAX_DRIVES) THEN
			CASE command OF

			1://Manual Reset
				ABB_EPL.Drives[belt].Manual.tof_run.IN := (velocity > 0);
				ABB_EPL.Drives[belt].Manual.Velocity := velocity;
				ABB_EPL.Drives[belt].Manual.Direction := direction;
			2: //Future Error Reset

			END_CASE;
			found := 1;
		ELSE
			error := 3;
		END_IF;

	ELSE
		error := 2;
	END_IF;

	sendResponse := (found > 0);
	errorResponse := (error > 0);

END_ACTION
```

#### _httpServer.st
```iecst
ACTION _httpServer:

	//Force the server to restart when then restart the PLC. Stops the server from crashing during PLC transfer
	IF (httpServer.status = ERR_FUB_ENABLE_FALSE) THEN
		httpServer.enable := 1;
	END_IF;
	//Error Handling -- Return the code 400 (Baf if there is a process error

	IF errorResponse THEN
		responseHeader.status := '400 Bad Request';
		sendResponse := 1;
	ELSIF ton_httpTimeOut.Q THEN
		responseHeader.status := '408 Request Timeout';
		responseData := 'Response Timeout';
		sendResponse := 1;
	ELSIF sendResponse THEN;
		responseHeader.status := '200 OK';
	END_IF;

	httpServer.enable := 1;
	httpServer.send := sendResponse; // Send Response on Rising edge.
	httpServer.abort := abortResponse;	//Send abort Response on Rising Edge

	IF (overRideData.responseDataLen > 0) THEN
		httpServer.responseDataLen := overRideData.responseDataLen;
	ELSE
		httpServer.responseDataLen := brsstrlen(ADR(responseData));
	END_IF;
	IF overRideData.responseHeader.contentType <> '' THEN
		responseHeader.contentType := overRideData.responseHeader.contentType;
	ELSIF overRideData.responseHeader.contentType <> 'nothing' THEN
		responseHeader.contentType := '';
	ELSE
		responseHeader.contentType := 'text/plain';
	END_IF;
	IF overRideData.responseHeader.status <> '' THEN
		responseHeader.status := overRideData.responseHeader.status;
	END_IF;

	responseHeader.contentLength := httpServer.responseDataLen;

	IF sendBinaryData THEN
		httpServer.pResponseData := ADR(responseDataBinary);
	ELSE
		httpServer.pResponseData := ADR(responseData);
	END_IF;
	httpServer();

	sendBinaryData := 0;

	IF (httpServer.phase = httpPHASE_RECEIVED) AND NOT sendResponse THEN
		recieved := 1;
	ELSE
		recieved := 0;
	END_IF;
	//Clear the overrides
	overRideData.responseDataLen 			:= 0;
	overRideData.responseHeader				:= BLANK_RESPONSE_HEADER;

	sendResponse := 0;
	abortResponse := 0;
	errorResponse := 0;

	//Request Timeout
	ton_httpTimeOut(IN:= (httpServer.phase = httpPHASE_RECEIVED),PT:= 500);//500
END_ACTION
```

#### _getLoadingData.st
```iecst
ACTION _getLoadingData:

	prg	:= 0;
	cat := 0;
	cus := 0;
	dst := 0;
	sp1 := 0;
	sp2 := 0;
	sp3 := 0;
	index 	:= 0;

	error := 0;
	found := 0;
	//Set common parameters of the function.
	getParameterName.searchString := requestData;
	getParameterName.searchOffset := 0;
	getParameterName.searchEndProperty := STRING_DOLLAR;

	//Find the id
	getParameterName.searchPropertyName := '"displayId":';
	getParameterName.searchEndProperty := ',';
	getParameterName();
	IF getParameterName.status = ERR_OK THEN
		index := DINT_TO_UDINT(atoi(ADR(getParameterName.outputValue)));
		getParameterName.searchOffset := getParameterName.nextPosition;
	ELSE
		error := 1;
	END_IF;

	//Find the category
	getParameterName.searchPropertyName := '"cat":';
	getParameterName.searchEndProperty := ',';
	getParameterName();
	IF getParameterName.status = ERR_OK THEN
		cat := DINT_TO_UDINT(atoi(ADR(getParameterName.outputValue)));
		getParameterName.searchOffset := getParameterName.nextPosition;
	ELSE
		error := 2;
	END_IF;

	//Find the customer
	getParameterName.searchPropertyName := '"cus":';
	getParameterName.searchEndProperty := ',';
	getParameterName();
	IF getParameterName.status = ERR_OK THEN
		cus := DINT_TO_UDINT(atoi(ADR(getParameterName.outputValue)));
		getParameterName.searchOffset := getParameterName.nextPosition;
	ELSE
		error := 3;
	END_IF;

	//Find the Program
	getParameterName.searchPropertyName := '"prg":';
	getParameterName.searchEndProperty := ',';
	getParameterName();
	IF getParameterName.status = ERR_OK THEN
		prg := DINT_TO_USINT(atoi(ADR(getParameterName.outputValue)));
		getParameterName.searchOffset := getParameterName.nextPosition;
	ELSE
		error := 5;
	END_IF;

	//Find the sp1
	getParameterName.searchPropertyName := '"sp1":';
	getParameterName.searchEndProperty := ',';
	getParameterName();
	IF getParameterName.status = ERR_OK THEN
		sp1 := DINT_TO_UINT(atoi(ADR(getParameterName.outputValue)));
		getParameterName.searchOffset := getParameterName.nextPosition;
	ELSE
		error := 6;
	END_IF;

	//Find the sp2
	getParameterName.searchPropertyName := '"sp2":';
	getParameterName.searchEndProperty := ',';
	getParameterName();
	IF getParameterName.status = ERR_OK THEN
		sp2 := DINT_TO_UINT(atoi(ADR(getParameterName.outputValue)));
		getParameterName.searchOffset := getParameterName.nextPosition;
	ELSE
		error := 7;
	END_IF;
	//Find the sp3
	getParameterName.searchPropertyName := '"sp3":';
	getParameterName.searchEndProperty := ',';
	getParameterName();
	IF getParameterName.status = ERR_OK THEN
		sp3 := DINT_TO_UINT(atoi(ADR(getParameterName.outputValue)));
		getParameterName.searchOffset := 0;
	ELSE
		error := 8;
	END_IF;

	//Find the program
	getParameterName.searchPropertyName := '"dst":';
	getParameterName.searchEndProperty := ',';
	getParameterName();
	IF getParameterName.status = ERR_OK THEN
		dst := DINT_TO_USINT(atoi(ADR(getParameterName.outputValue)));
		IF (index <= MAX_DISPLAYS) THEN
			found := found + 1;
			bag ACCESS ADR(LiveData_Recv[index].Bag);
			bag.Cat := cat;
			bag.Prg := prg;
			bag.Cus := cus;
			bag.Dst := dst;
			LiveData_Recv[index].Setpoints.SP1 := sp1 * 10;
			LiveData_Recv[index].Setpoints.SP2:= sp2 * 10;
			LiveData_Recv[index].Setpoints.SP3 := sp3 * 10;
		ELSE
			error := 99;
			overRideData.responseHeader.status := '404 Not Found';
			responseData := 'Unknown display';
			httpServer.responseDataLen := LEN(responseData);
		END_IF;
	ELSE
		error := 10;
	END_IF;

	sendResponse := (found > 0);
	errorResponse := (error > 0);

END_ACTION
```

#### _getLoadingSubmit.st
```iecst
ACTION _getLoadingSubmit:

	prg	:= 0;
	cat := 0;
	cus := 0;
	dst := 0;
	sp1 := 0;
	sp2 := 0;
	sp3 := 0;
	index 	:= 0;

	error := 0;
	found := 0;
	//Set common parameters of the function.
	getParameterName.searchString := requestData;
	getParameterName.searchOffset := 0;
	getParameterName.searchEndProperty := STRING_DOLLAR;

	//Find the index
	getParameterName.searchPropertyName := '"displayId":';
	getParameterName.searchEndProperty := ',';
	getParameterName();
	IF getParameterName.status = ERR_OK THEN
		index := DINT_TO_UDINT(atoi(ADR(getParameterName.outputValue)));
		getParameterName.searchOffset := getParameterName.nextPosition;
	ELSE
		error := 1;
	END_IF;

	//Find the category
	getParameterName.searchPropertyName := '"cat":';
	getParameterName.searchEndProperty := ',';
	getParameterName();
	IF getParameterName.status = ERR_OK THEN
		cat := DINT_TO_UDINT(atoi(ADR(getParameterName.outputValue)));
		getParameterName.searchOffset := getParameterName.nextPosition;
	ELSE
		error := 2;
	END_IF;

	//Find the customer
	getParameterName.searchPropertyName := '"cus":';
	getParameterName.searchEndProperty := ',';
	getParameterName();
	IF getParameterName.status = ERR_OK THEN
		cus := DINT_TO_UDINT(atoi(ADR(getParameterName.outputValue)));
		getParameterName.searchOffset := getParameterName.nextPosition;
	ELSE
		error := 3;
	END_IF;

	//Find the Program
	getParameterName.searchPropertyName := '"prg":';
	getParameterName.searchEndProperty := ',';
	getParameterName();
	IF getParameterName.status = ERR_OK THEN
		prg := DINT_TO_USINT(atoi(ADR(getParameterName.outputValue)));
		getParameterName.searchOffset := getParameterName.nextPosition;
	ELSE
		error := 5;
	END_IF;

	//Find the sp1
	getParameterName.searchPropertyName := '"sp1":';
	getParameterName.searchEndProperty := ',';
	getParameterName();
	IF getParameterName.status = ERR_OK THEN
		sp1 := DINT_TO_UINT(atoi(ADR(getParameterName.outputValue)));
		getParameterName.searchOffset := getParameterName.nextPosition;
	ELSE
		error := 6;
	END_IF;

	//Find the sp2
	getParameterName.searchPropertyName := '"sp2":';
	getParameterName.searchEndProperty := ',';
	getParameterName();
	IF getParameterName.status = ERR_OK THEN
		sp2 := DINT_TO_UINT(atoi(ADR(getParameterName.outputValue)));
		getParameterName.searchOffset := getParameterName.nextPosition;
	ELSE
		error := 7;
	END_IF;
	//Find the sp3
	getParameterName.searchPropertyName := '"sp3":';
	getParameterName.searchEndProperty := ',';
	getParameterName();
	IF getParameterName.status = ERR_OK THEN
		sp3 := DINT_TO_UINT(atoi(ADR(getParameterName.outputValue)));
		getParameterName.searchOffset := 0;
	ELSE
		error := 8;
	END_IF;

	//Find the program
	getParameterName.searchPropertyName := '"dst":';
	getParameterName.searchEndProperty := ',';
	getParameterName();
	IF getParameterName.status = ERR_OK THEN
		dst := DINT_TO_USINT(atoi(ADR(getParameterName.outputValue)));
		IF (index <= MAX_DISPLAYS) THEN
			found := found + 1;
			bag ACCESS ADR(LiveData_Recv[index].Bag);
			bag.Cat := cat;
			bag.Prg := prg;
			bag.Cus := cus;
			bag.Dst := dst;
			LiveData_Recv[index].Setpoints.SP1 := sp1 * 10;
			LiveData_Recv[index].Setpoints.SP2:= sp2 * 10;
			LiveData_Recv[index].Setpoints.SP3 := sp3 * 10;
			LiveData_Recv[index].Submit_Loading := 1;
		ELSE
			error := 99;
			overRideData.responseHeader.status := '404 Not Found';
			responseData := 'Unknown display';
			httpServer.responseDataLen := LEN(responseData);
		END_IF;
	ELSE
		error := 10;
	END_IF;

	sendResponse := (found > 0);
	errorResponse := (error > 0);

END_ACTION
```
